Yaskawa INFORM job: R2_O57-69(2)(90,180)OLD.JBI

/JOB
//NAME R2_O57-69(2)(90,180)OLD
//POS
///NPOS 642,642,642,18,0,0
///TOOL 0
///POSTYPE PULSE
///PULSE
C00000=-118942,38116,3308,-51577,58996,23781
C00001=-120746,43281,8706,-50981,57603,23623
C00002=-121445,45407,10966,-50768,57038,23575
C00003=-122175,45836,11424,-50421,56611,23420
C00004=-121445,45407,10966,-50768,57038,23575
C00005=-119713,46835,12049,-51615,58009,23970
C00006=-119593,49070,14464,-51837,57860,24140
C00007=-119713,46835,12049,-51615,58009,23970
C00008=-119003,44749,9818,-51825,58584,24014
C00009=-117170,39689,4492,-52413,60002,24162
C00010=-133704,84336,30677,-4045,90342,4182
C00011=-133972,88781,39264,-3963,87336,4193
C00012=-134077,90756,42954,-3934,86079,4199
C00013=-134077,90297,43636,-3936,85425,4220
C00014=-134077,90756,42954,-3934,86079,4199
C00015=-134064,91533,43556,-3938,86108,4203
C00016=-134173,94225,46985,-3908,85378,4191
C00017=-134064,91533,43556,-3938,86108,4203
C00018=-133960,89550,39850,-3967,87371,4196
C00019=-133691,85093,31233,-4049,90389,4184
C00020=-133097,85072,31507,-9968,91856,10528
C00021=-133756,89066,39535,-9767,88935,10550
C00022=-134013,90847,42981,-9696,87717,10563
C00023=-134013,90387,43661,-9698,87071,10613
C00024=-134013,90847,42981,-9696,87717,10563
C00025=-134077,91446,43535,-9678,87677,10545
C00026=-134345,93924,46689,-9607,86989,10512
C00027=-134077,91446,43535,-9678,87677,10545
C00028=-133821,89654,40071,-9749,88900,10532
C00029=-133165,85640,32010,-9949,91831,10509
C00030=-130607,9372,-15044,-13437,81583,13219
C00031=-132164,5171,-3952,-15307,72023,14325
C00032=-104612,24784,65967,-49840,36559,34272
C00033=-106530,34976,78845,-52404,33899,35280
C00034=-107268,39847,85132,-53931,32696,35940
C00035=-107268,43497,90995,-56192,31674,37136
C00036=-107268,39847,85132,-53931,32696,35940
C00037=-106991,38998,84230,-53831,32905,35947
C00038=-107592,41782,87346,-54342,32315,36087
C00039=-106991,38998,84230,-53831,32905,35947
C00040=-106248,34218,78071,-52358,34091,35316
C00041=-104315,24157,65380,-49864,36729,34346
C00042=-95633,-69755,-51009,-37313,58213,27375
C00043=-82988,-118583,-84497,-42047,60487,32680
C00044=-200995,-130184,-93319,70720,78040,-43840
C00045=-163099,-71600,-71646,60941,59675,-30655
C00046=-151416,29115,15831,69500,88499,-38418
C00047=-148764,29488,16198,69305,86698,-38096
C00048=-147706,29711,16418,69221,85978,-37969
C00049=-147097,31186,17883,69177,85514,-37952
C00050=-147706,29711,16418,69221,85978,-37969
C00051=-147508,26891,13470,69190,85984,-37787
C00052=-146989,25154,11784,69139,85690,-37658
C00053=-147508,26891,13470,69190,85984,-37787
C00054=-148579,26663,13248,69280,86712,-37916
C00055=-151265,26278,12874,69491,88533,-38244
C00056=-151230,28714,15393,69487,88397,-38368
C00057=-148574,29104,15777,69288,86594,-38045
C00058=-147514,29335,16004,69203,85873,-37918
C00059=-146906,30812,17468,69159,85409,-37901
C00060=-147514,29335,16004,69203,85873,-37918
C00061=-147724,26972,13590,69210,86117,-37828
C00062=-147207,25230,11899,69159,85824,-37699
C00063=-147724,26972,13590,69210,86117,-37828
C00064=-148795,26752,13377,69299,86844,-37957
C00065=-151480,26388,13023,69506,88665,-38286
C00066=-150499,113686,46157,71277,96983,-27560
C00067=-148414,114188,46840,70516,95698,-27414
C00068=-147582,114456,47206,70210,95177,-27363
C00069=-147103,116179,49560,69975,94689,-27557
C00070=-147582,114456,47206,70210,95177,-27363
C00071=-147564,110815,41655,70398,95727,-26688
C00072=-147157,108917,39076,70325,95714,-26378
C00073=-147564,110815,41655,70398,95727,-26688
C00074=-148407,110561,41310,70722,96244,-26740
C00075=-150520,110089,40669,71527,97523,-26888
C00076=-135781,-39109,-42450,-5820,71469,-27792
C00077=-134852,-34609,-36187,-6165,70004,-27387
C00078=-134494,-32781,-33633,-6302,69403,-27227
C00079=-134494,-32513,-32201,-6332,68664,-27188
C00080=-134494,-32781,-33633,-6302,69403,-27227
C00081=-134576,-33268,-34172,-6273,69478,-27261
C00082=-134372,-31123,-32745,-6329,69716,-27200
C00083=-134576,-33268,-34172,-6273,69478,-27261
C00084=-133492,-33488,-34057,-6622,69381,-26865
C00085=-132368,-33840,-34288,-6976,69438,-26463
C00086=-133492,-33488,-34057,-6622,69381,-26865
C00087=-133841,-35331,-36614,-6487,69976,-27023
C00088=-134747,-39871,-42887,-6148,71424,-27423
C00089=-122053,-39806,-42652,-15420,62809,-34817
C00090=-121499,-35034,-36226,-15868,61466,-34410
C00091=-121286,-33103,-33607,-16052,60912,-34244
C00092=-121286,-32828,-32171,-16165,60197,-34138
C00093=-121286,-33103,-33607,-16052,60912,-34244
C00094=-121314,-33263,-34344,-15985,61264,-34307
C00095=-121302,-31081,-32892,-15957,61485,-34335
C00096=-121314,-33263,-34344,-15985,61264,-34307
C00097=-119787,-33398,-34061,-16683,61335,-33713
C00098=-118651,-33362,-34037,-17169,61575,-33298
C00099=-119787,-33398,-34061,-16683,61335,-33713
C00100=-119983,-35334,-36680,-16506,61888,-33874
C00101=-120494,-40120,-43107,-16077,63224,-34271
C00102=-114895,-27674,-41035,-24554,79329,-24611
C00103=-103160,-731,-14280,-43401,100853,-1823
C00104=-105135,1502,-9443,-43163,98538,-1741
C00105=-105913,2477,-7430,-43084,97612,-1705
C00106=-105914,2666,-6021,-42996,97041,-1463
C00107=-105913,2477,-7430,-43084,97612,-1705
C00108=-127520,-68112,-41549,-19229,27618,7061
C00109=-127380,-66019,-40542,-19113,28083,7011
C00110=-127520,-68112,-41549,-19229,27618,7061
C00111=-133514,-23938,-39247,-1523,83124,-19162
C00112=-132464,-24298,-39502,-1762,83117,-18812
C00113=-133514,-23938,-39247,-1523,83124,-19162
C00114=-133840,-25466,-41668,-1447,83823,-19278
C00115=-134685,-29188,-47604,-1253,85549,-19576
C00116=-94540,-44906,-54644,-54690,80182,11416
C00117=-2997,-159102,-96620,-35577,110249,43089
C00118=-94928,-31896,-36448,-44981,51726,73410
C00119=-97674,-28950,-32085,-44251,49500,73032
C00120=-98746,-27702,-30280,-43966,48623,72882
C00121=-98747,-27457,-28859,-44425,48077,73195
C00122=-98746,-27702,-30280,-43966,48623,72882
C00123=-99145,-25229,-28534,-43633,48570,72671
C00124=-99641,-23313,-27181,-43273,48438,72445
C00125=-99145,-25229,-28534,-43633,48570,72671
C00126=-99389,-27279,-29944,-43614,48313,72668
C00127=-100362,-28273,-30629,-43136,47769,72383
C00128=-99389,-27279,-29944,-43614,48313,72668
C00129=-98324,-28543,-31764,-43902,49185,72819
C00130=-95596,-31533,-36163,-44641,51397,73201
C00131=-73206,-49255,-47301,-54380,62174,80035
C00132=-83647,-21856,-29546,-43638,51559,72523
C00133=-86196,-18896,-25023,-42989,49379,72216
C00134=-87192,-17643,-23150,-42742,48516,72095
C00135=-87193,-17430,-21742,-43197,47953,72406
C00136=-87192,-17643,-23150,-42742,48516,72095
C00137=-87217,-17769,-23202,-42747,48480,72100
C00138=-88162,-16936,-22585,-42189,48060,71766
C00139=-87217,-17769,-23202,-42747,48480,72100
C00140=-86221,-19023,-25076,-42995,49342,72221
C00141=-83670,-21988,-29600,-43645,51522,72530
C00142=-60313,-109588,-73152,-60260,62863,-74993
C00143=-60313,-109588,-73152,-60260,62863,-74993
C00144=-60313,-109588,-73152,-60260,62863,-74993
C00145=-60313,-109588,-73152,-60260,62863,-74993
C00146=-121468,-98128,-128632,1200,91954,-4785
C00147=-120935,-89040,-122262,1025,92698,-4621
C00148=-120739,-85841,-119804,961,92827,-4562
C00149=-120740,-85741,-118114,960,91838,-4570
C00150=-120739,-85841,-119804,961,92827,-4562
C00151=-120638,-81288,-118578,930,94411,-4521
C00152=-120241,-74983,-116497,803,96366,-4393
C00153=-120638,-81288,-118578,930,94411,-4521
C00154=-120828,-84219,-120984,993,94387,-4576
C00155=-121344,-92430,-127180,1163,93987,-4729
C00156=-126619,-93375,-85777,19436,85602,-57728
C00157=-123229,-93449,-82463,19138,82838,-56953
C00158=-121861,-93330,-81074,19019,81766,-56629
C00159=-121850,-91527,-78779,19037,81304,-56698
C00160=-121861,-93330,-81074,19019,81766,-56629
C00161=-120032,-93477,-81181,18813,81333,-56039
C00162=-117985,-95044,-81508,18598,80291,-55463
C00163=-120032,-93477,-81181,18813,81333,-56039
C00164=-121407,-93650,-82591,18940,82390,-56369
C00165=-124815,-93717,-85961,19254,85118,-57161
C00166=-105133,-95150,-84366,-27685,77771,48864
C00167=-109419,-93151,-80804,-27043,75322,47788
C00168=-111110,-92231,-79325,-26774,74383,47352
C00169=-111209,-90435,-77025,-26813,73909,47425
C00170=-111110,-92231,-79325,-26774,74383,47352
C00171=-111989,-92454,-79471,-26607,74078,47081
C00172=-114284,-92810,-79614,-26159,73263,46376
C00173=-111989,-92454,-79471,-26607,74078,47081
C00174=-110299,-93409,-80962,-26883,75006,47521
C00175=-106012,-95496,-84557,-27540,77427,48607
C00176=-111909,-102425,-108765,-17811,80188,32257
C00177=-116710,-109323,-114600,-10394,73642,20182
C00178=-119128,-100378,-108798,-9411,74366,19294
C00179=-120024,-97049,-106503,-9050,74562,18974
C00180=-120031,-96065,-104948,-9065,74116,19005
C00181=-120024,-97049,-106503,-9050,74562,18974
C00182=-121130,-95394,-105931,-8599,74938,18572
C00183=-122871,-95322,-105904,-7915,74788,17994
C00184=-121130,-95394,-105931,-8599,74938,18572
C00185=-120110,-94835,-105770,-8990,75231,18895
C00186=-120119,-91118,-104720,-8941,76480,18801
C00187=-120110,-94835,-105770,-8990,75231,18895
C00188=-119227,-98081,-108057,-9343,75070,19206
C00189=-116847,-106779,-113833,-10301,74448,20066
C00190=-125162,-107696,-115002,11574,77940,-27023
C00191=-122232,-100471,-109587,10556,77926,-26035
C00192=-121132,-97724,-107430,10172,77873,-25669
C00193=-121129,-96411,-105359,10192,77282,-25717
C00194=-121132,-97724,-107430,10172,77873,-25669
C00195=-120375,-94991,-106195,9888,78418,-25371
C00196=-118057,-94902,-106157,9076,78179,-24616
C00197=-120375,-94991,-106195,9888,78418,-25371
C00198=-121123,-94352,-106931,10125,79277,-25551
C00199=-121107,-89294,-105478,10075,80954,-25409
C00200=-121123,-94352,-106931,10125,79277,-25551
C00201=-122203,-96975,-109071,10499,79378,-25901
C00202=-125076,-103844,-114435,11488,79527,-26845
C00203=-120615,-96693,-99705,24269,61927,-46070
C00204=-120615,-96754,-97435,24583,60621,-46372
C00205=-120615,-96734,-96510,24712,60111,-46493
C00206=-120613,-97925,-98139,24620,60467,-46408
C00207=-122356,-96694,-96496,25580,60643,-47091
C00208=-120617,-95462,-105609,23301,89319,-42487
C00209=-120616,-96376,-102090,23303,86889,-42960
C00210=-120616,-96174,-102896,20314,113785,-36834
C00211=-120616,-95912,-104039,20462,114573,-36686
C00212=-120617,-94981,-106794,20878,116613,-36292
C00213=-120641,-102950,-117078,-2305,90642,6155
C00214=-120615,-96500,-96704,-24731,54164,47412
C00215=-120614,-96434,-94585,-25118,53008,47710
C00216=-120614,-96374,-93724,-25277,52554,47829
C00217=-118876,-96339,-93708,-26332,53098,48481
C00218=-120612,-97606,-95370,-25157,52900,47739
C00219=-120617,-94939,-106140,-23447,89820,42327
C00220=-120616,-95118,-105679,-23443,89475,42395
C00221=-120617,-94553,-107144,-21169,116976,36148
C00222=-120617,-94008,-108179,-21364,117834,35974
C00223=-120617,-92305,-110644,-21913,120064,35505
C00224=-120658,-79064,-115821,-20777,115116,36511
C00225=-120619,-89788,-115023,8813,72744,77332
C00226=-120618,-92923,-112261,8977,69472,77088
C00227=-120618,-93918,-111063,9048,68239,76994
C00228=-120616,-94647,-112535,9016,68763,77035
C00229=-120317,-89862,-109879,8813,69547,77195
C00230=-120618,-93982,-110933,9081,68131,76955
C00231=-120618,-94046,-110802,9114,68024,76915
C00232=-120618,-94709,-109820,9197,65184,76768
C00233=-120617,-95196,-108972,8506,62672,76659
C00234=-120617,-95481,-108396,7103,60843,76635
C00235=-120617,-95545,-108232,5697,60110,76679
C00236=-120618,-93518,-111355,4944,62938,76697
C00237=-120618,-93446,-111427,4025,62977,76727
C00238=-120618,-93195,-111705,2442,63558,76792
C00239=-120618,-92705,-112237,841,64979,76863
C00240=-120618,-92008,-112941,-348,67067,76917
C00241=-120618,-91373,-113529,-886,68931,76945
C00242=-120619,-90404,-114488,-945,70932,76821
C00243=-120619,-89573,-115103,-879,73169,76864
C00244=-120619,-88566,-115779,-154,75847,76963
C00245=-120619,-87861,-116220,1182,77795,77117
C00246=-120619,-87671,-116345,2465,78546,77256
C00247=-120619,-91363,-113807,3286,75243,77100
C00248=-120619,-91437,-113755,4139,75204,77156
C00249=-120618,-91668,-113564,5199,74797,77209
C00250=-120618,-91861,-113400,6010,74299,77242
C00251=-120618,-92325,-112970,7121,73103,77250
C00252=-120618,-92854,-112432,8036,71559,77218
C00253=-120618,-93200,-112056,8504,70412,77180
C00254=-120618,-93741,-111409,8966,68528,77095
C00255=-120618,-93842,-111215,9015,68365,77035
C00256=-120618,-93908,-111085,9047,68257,76996
C00257=-120618,-92911,-112281,8976,69491,77090
C00258=-120619,-89769,-115041,8812,72765,77333
C00259=-120613,-94111,-83344,23310,76872,-48529
C00260=-120612,-93123,-79966,23449,75424,-48818
C00261=-120612,-92685,-78593,23509,74854,-48933
C00262=-120519,-94136,-80334,23460,75127,-48843
C00263=-122104,-91474,-78326,23730,75702,-49326
C00264=-117316,-93808,-82805,15952,85371,-55800
C00265=-120612,-92504,-78008,16222,83828,-57165
C00266=-120612,-92225,-77144,16221,83447,-57214
C00267=-120612,-92754,-78742,16205,84132,-57123
C00268=-120612,-93939,-82668,16176,85870,-56895
C00269=-114287,-94620,-89520,-6331,89004,4508
C00270=-108926,-90943,-77088,-25317,82681,56680
C00271=-112815,-90510,-73836,-25087,79880,55819
C00272=-114383,-90199,-72475,-24991,78788,55461
C00273=-114333,-91608,-74232,-24970,79128,55408
C00274=-112663,-89963,-72378,-25142,79365,55987
C00275=-114583,-88799,-68791,-27921,64605,46597
C00276=-114487,-93503,-82637,-26827,70088,45260
C00277=-115264,-91797,-76742,-30984,57662,33422
C00278=-113792,-91904,-77552,-31424,58590,33801
C00279=-110138,-91921,-79470,-32448,60976,34690
C00280=-60313,-109588,-73152,-60260,62863,-74993
C00281=-60313,-109588,-73152,-60260,62863,-74993
C00282=-60313,-109588,-73152,-60260,62863,-74993
C00283=-60313,-109588,-73152,-60260,62863,-74993
C00284=-93056,-22452,-26427,-62683,51364,-68554
C00285=-94918,-23815,-27400,-62098,50128,-68890
C00286=-95672,-24335,-27768,-61852,49629,-69030
C00287=-95671,-24543,-29165,-61297,50004,-69420
C00288=-95119,-26190,-29068,-62168,49906,-68831
C00289=-113833,-31923,-32981,-19338,22123,-69808
C00290=-113432,-31852,-32933,-20038,22233,-69480
C00291=-111211,-31381,-32618,-29195,23933,-65184
C00292=-107573,-30332,-31913,-37350,26359,-61322
C00293=-106073,-29797,-31550,-41773,28129,-59204
C00294=-102671,-28354,-30566,-47316,31086,-56518
C00295=-101245,-27653,-30084,-50385,33119,-55008
C00296=-96015,-24564,-27929,-57391,39606,-51469
C00297=-95870,-24466,-27860,-57479,39693,-51427
C00298=-98425,-26093,-29002,-49127,35298,-40867
C00299=-98535,-26162,-29051,-49050,35234,-40906
C00300=-98812,-26334,-29170,-48853,35075,-41005
C00301=-94260,-52437,-45641,-55679,35604,-37348
C00302=-53363,-13156,-19582,-69042,101484,-57693
C00303=-70300,5852,-4038,-68507,90193,-60008
C00304=-72032,2742,-6705,-68392,89052,-60255
C00305=-72741,1528,-7732,-68341,88581,-60353
C00306=-72740,1358,-9123,-68348,88884,-60681
C00307=-71868,858,-8294,-68404,89165,-60238
C00308=-77282,-5546,-13564,-65427,71560,-48018
C00309=-76174,-3931,-12256,-66124,74358,-47138
C00310=-77728,-6177,-14071,-64696,69365,-41232
C00311=-76987,-5122,-13221,-65187,71135,-40572
C00312=-78162,-6780,-14553,-64908,67376,-44626
C00313=-76574,-4519,-12734,-65439,69183,-44207
C00314=-75699,-3215,-11672,-66019,71276,-43722
C00315=-73856,-322,-9283,-66697,73982,-43118
C00316=-73074,967,-8204,-67155,75992,-42677
C00317=-72162,2519,-6894,-67667,78480,-42145
C00318=-70374,5730,-4143,-68213,81550,-41494
C00319=-70642,5234,-4572,-68092,80748,-41661
C00320=-70220,6012,-3899,-68142,81024,-41598
C00321=-69181,7983,-2180,-68262,81700,-41439
C00322=-53363,-13156,-19582,-69042,101484,-57693
C00323=-88855,-179547,-122665,-16422,45831,14756
C00324=-103013,-99268,-100595,-7137,71031,6353
C00325=-111832,16928,28851,-4518,50540,4019
C00326=-112106,24952,39258,-4538,48250,4007
C00327=-112211,28376,43752,-4558,47241,4009
C00328=-112092,25909,41315,-4600,47479,4051
C00329=-112213,27385,41422,-4491,48163,3964
C00330=-110994,29129,44722,-10026,47870,8913
C00331=-107882,31558,47633,-16852,48960,15049
C00332=-106420,34221,50265,-20220,50689,15733
C00333=-107556,33681,49588,-20659,51389,16328
C00334=-107303,34756,50847,-23620,53119,19537
C00335=-105809,38630,55063,-26127,54547,25185
C00336=-100600,65185,87794,-37926,61057,39597
C00337=-99799,61843,82703,-37497,62519,39384
C00338=-97770,55081,72181,-36715,65773,39058
C00339=-113055,9147,22486,-11521,49710,9806
C00340=-113748,16710,31984,-11522,47692,9742
C00341=-114014,19893,36035,-11546,46813,9730
C00342=-113504,17960,34216,-11778,47009,9938
C00343=-114013,18924,33775,-11384,47689,9622
C00344=-106504,35034,50196,-27270,57817,24489
C00345=-107808,31596,46678,-26860,57759,23943
C00346=-101619,66436,89448,-39641,65847,43373
C00347=-100773,63725,85128,-39270,67197,43204
C00348=-98646,58275,76145,-38555,70253,42947
C00349=-99884,14179,20835,-32070,74790,34547
C00350=-104259,-119010,-113397,-13066,68419,11198
C00351=-100618,-153040,-123102,-15914,57898,13971
C00352=-171047,-67517,-68920,2824,104590,-81494
C00353=-162612,-44481,-56179,3922,108231,-78415
C00354=-172950,15898,5057,-12161,117913,80240
C00355=-173383,11030,3410,-12137,116393,80239
C00356=-173563,9131,2831,-12130,115759,80238
C00357=-174118,10117,2984,-12376,116079,79984
C00358=-173005,10826,4333,-11924,115790,80453
C00359=-173900,36762,39678,-14923,122347,88654
C00360=-174631,19304,16630,-12631,116903,82099
C00361=-174582,11977,8086,-12295,113872,80049
C00362=-174393,13825,8643,-12294,114494,80054
C00363=-173937,18573,10240,-12297,115988,80066
C00364=-161354,27343,19699,-12039,109597,67520
C00365=-162299,23506,18954,-12170,107974,67338
C00366=-162689,22031,18738,-12226,107304,67264
C00367=-162689,21613,17076,-12289,108094,67181
C00368=-162258,23995,20616,-12099,107225,67431
C00369=-160599,18374,15454,-16346,104951,65883
C00370=-160862,19037,16144,-16128,105227,62268
C00371=-158963,16179,14200,-19810,103313,58208
C00372=-158332,17222,14010,-19745,104082,58313
C00373=-156794,20003,13731,-19594,105963,58572
C00374=-161333,16594,8144,-10689,103467,-23902
C00375=-160995,17911,13523,-10509,100921,-23559
C00376=-160860,18544,15785,-10444,99888,-23423
C00377=-160126,17389,14600,-10331,100117,-23184
C00378=-160925,18232,14234,-10487,100661,-23512
C00379=-160747,19067,16273,-10425,99872,-23382
C00380=-160882,18430,14006,-10490,100906,-23518
C00381=-161218,17106,8616,-10669,103455,-23860
C00382=-159736,50763,37041,-6948,117736,-78214
C00383=-159788,45167,33757,-6909,116883,-78180
C00384=-159810,42990,32553,-6892,116506,-78165
C00385=-160346,43786,32675,-7123,116791,-78393
C00386=-159444,45178,34878,-6729,116233,-78006
C00387=-161348,81543,87740,-6707,117550,-69501
C00388=-161230,54566,49708,-6566,116296,-76295
C00389=-160797,45806,38282,-7135,114356,-78411
C00390=-160766,47971,39500,-7147,114719,-78422
C00391=-160691,53556,42838,-7172,115535,-78445
C00392=-154706,39789,27555,-8539,114606,12724
C00393=-148495,53758,55593,-7913,102792,72747
C00394=-149088,49534,53986,-8041,101563,72620
C00395=-149332,47922,53457,-8093,101041,72570
C00396=-149332,46980,51118,-8127,101987,72507
C00397=-149055,50602,56404,-8000,100635,72693
C00398=-147241,44754,50188,-12563,99747,71321
C00399=-147513,45427,50986,-12280,99912,67703
C00400=-145634,43287,49424,-16194,98869,63733
C00401=-145156,44506,49535,-16105,99500,63818
C00402=-143994,47742,50063,-15894,101016,64033
C00403=-161265,51089,39840,-10591,101724,-23724
C00404=-160975,52973,46100,-10427,98924,-23381
C00405=-160859,53890,48805,-10368,97764,-23243
C00406=-160229,52461,47107,-10276,98151,-23055
C00407=-160915,53398,46988,-10405,98609,-23333
C00408=-160762,54537,49526,-10349,97667,-23200
C00409=-160878,53605,46802,-10407,98831,-23339
C00410=-161167,51693,40503,-10570,101641,-23682
C00411=-148526,37088,19319,-8739,116408,71765
C00412=-149143,32311,17412,-8825,115075,71633
C00413=-149398,30453,16735,-8860,114515,71580
C00414=-149398,30263,15299,-8924,115292,71518
C00415=-149109,32604,18884,-8755,114332,71704
C00416=-147222,27780,14258,-13593,112811,69882
C00417=-147505,28304,14841,-13306,113042,66284
C00418=-145549,26214,13499,-17411,111682,61933
C00419=-145053,27746,13857,-17364,112331,62024
C00420=-143846,31723,14951,-17251,113896,62249
C00421=-164842,-38441,-59879,14258,84390,68161
C00422=-159089,-119441,-87904,20108,53110,65909
C00423=-167794,-136231,-92390,25307,50039,61231
C00424=-105945,-102671,-115440,26558,80933,-73598
C00425=-110364,-40123,-85663,27999,94589,-71935
C00426=-95866,64314,90102,38927,85041,-69053
C00427=-95118,63196,89692,39138,84476,-68962
C00428=-95722,60422,85500,38938,85635,-68779
C00429=-95367,67809,95356,39124,83704,-69344
C00430=-95389,64313,91842,39100,84004,-69244
C00431=-93119,49699,70965,34888,83296,-74684
C00432=-91573,45828,64995,32087,82929,-76236
C00433=-92175,46461,64458,31959,83708,-76245
C00434=-93644,48287,63421,31668,85593,-76279
C00435=-107566,-14252,9731,28298,67477,41115
C00436=-107311,-10314,17293,28810,65069,40577
C00437=-107211,-8617,20467,29042,64083,40348
C00438=-106149,-8342,20561,28950,63805,40701
C00439=-107303,-9723,18207,28865,64837,40517
C00440=-107260,-8071,20895,29042,64114,40337
C00441=-107361,-9770,17714,28809,65103,40566
C00442=-107614,-13711,10138,28297,67517,41106
C00443=-102856,-73680,-76596,22146,63215,42111
C00444=-159709,-90647,-84021,39939,81385,24012
C00445=-89629,-138278,-77876,-2613,32114,-4559
C00446=-116866,-116923,-63332,14121,27231,-27701
C00447=-115505,-113884,-61604,12498,27509,-26695
C00448=-115326,-115959,-62110,12631,26745,-26737
C00449=-117688,-114707,-62647,14613,28063,-28063
C00450=-116558,-113464,-61851,14335,28746,-26693
C00451=-118841,-112467,-62256,17923,31430,-26552
C00452=-113340,-111890,-64159,7172,33609,-21208
C00453=-114395,-115039,-66037,8124,33246,-21857
C00454=-122649,-85452,-63239,9213,34716,17761
C00455=-134041,-32885,-33620,13278,27002,71259
C00456=-134041,-32878,-33615,13278,27003,71259
C00457=-134041,-32875,-33613,13278,27003,71259
C00458=-134243,-35023,-35024,13683,26807,71061
C00459=-134041,-33117,-35025,12952,27729,71423
C00460=-134039,-32852,-33598,169,25633,78300
C00461=-134039,-32854,-33600,1649,26450,70781
C00462=-134033,-32782,-33552,-26231,28846,72528
C00463=-134032,-32780,-33551,-26232,28846,72529
C00464=-134031,-32775,-33547,-26233,28847,72529
C00465=-134045,-33787,-47185,-21244,36087,69888
C00466=-134041,-32886,-33621,13278,27002,71259
C00467=-134041,-32878,-33616,13278,27003,71259
C00468=-134041,-32875,-33614,13278,27003,71259
C00469=-134243,-35024,-35024,13684,26807,71061
C00470=-134041,-33118,-35026,12952,27729,71423
C00471=-134039,-32851,-33598,169,25633,78300
C00472=-134038,-32847,-33595,-898,26468,70800
C00473=-134033,-32781,-33552,-26231,28846,72528
C00474=-134032,-32780,-33550,-26232,28846,72529
C00475=-134031,-32775,-33547,-26233,28847,72529
C00476=-134033,-32807,-33569,-26308,35204,-51674
C00477=-134033,-32800,-33564,-26308,35204,-51674
C00478=-134033,-32797,-33562,-26308,35205,-51674
C00479=-134234,-34945,-34973,-26254,34929,-51698
C00480=-134032,-33039,-34974,-25852,35877,-51926
C00481=-134031,-32780,-33551,-33925,38137,-46837
C00482=-134030,-32755,-33534,-40499,34489,-51688
C00483=-134024,-32674,-33480,-63182,37461,-51745
C00484=-134024,-32672,-33479,-63182,37461,-51745
C00485=-134023,-32667,-33476,-63182,37462,-51745
C00486=-132274,-93805,-93411,-10969,51655,-47542
C00487=-128603,-177588,-92922,79935,27094,-30929
C00488=-220712,-98286,-76285,54391,96146,-31963
C00489=-184952,-63059,-48640,55161,75645,-24408
C00490=-160799,-33037,-33731,39953,86010,-17371
C00491=-160797,-33031,-33727,39953,86010,-17370
C00492=-161372,-34916,-34964,40000,86113,-17582
C00493=-161596,-32269,-33940,40001,86782,-17427
C00494=-160797,-33031,-33727,39954,86007,-17369
C00495=-160797,-33031,-33727,39954,86007,-17369
C00496=-160798,-33031,-33727,39953,86010,-17370
C00497=-160800,-33038,-33732,39953,86010,-17371
C00498=-161845,-54729,-47543,46717,77238,-21379
C00499=-134060,-33141,-33790,36180,74127,-10109
C00500=-134059,-33123,-33778,36179,74128,-10108
C00501=-134058,-33115,-33773,36179,74129,-10108
C00502=-134260,-35264,-35181,36258,74021,-10232
C00503=-134971,-32933,-34372,36300,74891,-10239
C00504=-134058,-33116,-33773,36179,74126,-10108
C00505=-134058,-33116,-33773,36179,74126,-10108
C00506=-134059,-33117,-33774,36179,74129,-10108
C00507=-134059,-33124,-33779,36179,74129,-10109
C00508=-134061,-33143,-33791,36180,74127,-10110
C00509=-154603,-70143,-52801,41434,56822,-11271
C00510=-233697,-158912,-98343,45711,85738,-36562
C00511=-192750,-134368,-116228,45795,59274,-21429
C00512=-146286,5957,-20405,4483,81226,-784
C00513=-143087,77833,55626,3655,71235,-21
C00514=-143077,84404,30410,3488,90094,518
C00515=-142973,88921,39083,3455,87079,467
C00516=-142932,90928,42809,3445,85817,446
C00517=-142932,91423,42172,3444,86463,463
C00518=-142895,88300,39491,3433,86507,476
C00519=-141651,91294,43270,3060,85682,850
C00520=-137685,92968,45398,1861,85119,2101
C00521=-140907,91434,44974,10035,83374,-9634
C00522=-141153,89375,41251,10096,84618,-9613
C00523=-141784,84734,32608,10277,87581,-9573
C00524=-134927,82297,28432,-4231,89843,4215
C00525=-135205,86732,36934,-4146,86884,4227
C00526=-135312,88694,40576,-4116,85649,4233
C00527=-135048,86331,37610,-4195,86271,4296
C00528=-135312,89191,39937,-4114,86296,4212
C00529=-131131,97718,51799,-14741,88225,12517
C00530=-134404,91131,43379,-13932,89423,11301
C00531=-135590,89058,40758,-13635,89764,10876
C00532=-135274,87435,37525,-13726,90938,10849
C00533=-134466,83798,29971,-13984,93767,10791
C00534=-124065,29550,-6223,-11945,87688,10852
C00535=-142798,-17443,-24047,-1901,70629,2085
C00536=-128958,-75577,-89763,-14465,60088,17152
C00537=-136794,-169084,-119686,-16507,29987,18519
C00538=-120728,-100182,-87766,90,59287,81758
C00539=-120667,-32765,-33541,61,60559,81782
C00540=-120668,-32752,-33532,62,60561,81781
C00541=-120669,-32746,-33528,62,60561,81781
C00542=-119537,-32735,-33521,-457,60565,82216
C00543=-120668,-32988,-34940,61,61306,81782
C00544=-120669,-32746,-33528,62,60561,81781
C00545=-120668,-32752,-33532,62,60561,81781
C00546=-120667,-32765,-33541,61,60559,81782
C00547=-129245,32742,-1401,19411,96333,49090
C00548=-120680,47311,12786,22923,98876,42875
C00549=-120681,47325,12802,22923,98874,42874
C00550=-120681,47331,12808,22923,98874,42874
C00551=-119944,47335,12813,22855,98676,43099
C00552=-120681,47590,11836,22981,99550,43006
C00553=-120681,47331,12808,22923,98874,42874
C00554=-120681,47325,12802,22923,98874,42874
C00555=-120680,47311,12786,22923,98876,42875
C00556=-120680,47311,12786,22923,98876,42875
C00557=-120681,47325,12802,22923,98874,42874
C00558=-120681,47331,12808,22923,98874,42874
C00559=-119944,47336,12814,22855,98676,43099
C00560=-120681,47591,11836,22981,99550,43006
C00561=-120681,47331,12808,22923,98874,42874
C00562=-120681,47325,12802,22923,98874,42874
C00563=-120680,47311,12786,22923,98876,42875
C00564=-130279,10433,-22592,19638,98058,49014
C00565=-80524,6289,-12410,27994,97930,43132
C00566=-80528,6302,-12399,27994,97931,43130
C00567=-80529,6307,-12395,27994,97931,43130
C00568=-80528,6342,-13609,28061,98610,43296
C00569=-80526,8467,-10508,27990,97885,43120
C00570=-80531,6315,-12388,27994,97932,43129
C00571=-80530,6310,-12392,27994,97931,43130
C00572=-80526,6297,-12403,27994,97930,43131
C00573=-80535,6328,-12377,43448,96376,44223
C00574=-80540,6344,-12363,43448,96378,44221
C00575=-80541,6350,-12357,43448,96378,44221
C00576=-80540,6385,-13571,43530,96942,44464
C00577=-80538,8511,-10470,43443,96339,44205
C00578=-80543,6359,-12350,43448,96379,44220
C00579=-80542,6352,-12355,43448,96378,44221
C00580=-80537,6336,-12370,43448,96376,44222
C00581=-80544,6364,-12345,43448,96379,44220
C00582=-80548,6380,-12331,43448,96381,44219
C00583=-80550,6387,-12325,43449,96382,44218
C00584=-80549,6422,-13539,43530,96945,44461
C00585=-80546,8548,-10438,43443,96342,44203
C00586=-80552,6395,-12318,43449,96383,44218
C00587=-80550,6388,-12324,43449,96382,44218
C00588=-80545,6372,-12338,43448,96380,44220
C00589=-80549,-32984,-33707,19991,70236,-81341
C00590=-80555,-32968,-33696,19993,70239,-81342
C00591=-80557,-32962,-33692,19994,70240,-81343
C00592=-80555,-33203,-35103,19909,70941,-81221
C00593=-80552,-30784,-32238,19966,70451,-81305
C00594=-80559,-32953,-33686,19994,70241,-81344
C00595=-80557,-32960,-33690,19994,70240,-81343
C00596=-80551,-32976,-33701,19992,70237,-81341
C00597=-125854,-89644,-68041,26288,64871,-64769
C00598=-122217,-87418,-63795,25670,62409,-63867
C00599=-120772,-86435,-62049,25411,61450,-63497
C00600=-122467,-86560,-62389,25830,62102,-64046
C00601=-120772,-87141,-63633,25274,62005,-63363
C00602=-120758,-81751,-60100,25140,62542,-63230
C00603=-120623,13667,2850,23403,71928,-61123
C00604=-120620,18086,6907,23432,71720,-61165
C00605=-121318,17638,5194,23528,72676,-61236
C00606=-123068,16745,1131,23791,75052,-61411
C00607=-120718,-27867,-44657,79,69917,81769
C00608=-120718,-26776,-39817,80,67499,81767
C00609=-120718,-26257,-37822,80,66538,81767
C00610=-119640,-26248,-37815,-390,66541,82155
C00611=-120717,-26264,-39071,80,67303,81767
C00612=-120711,-21841,-34695,77,66883,81769
C00613=-120650,35351,15016,51,65678,81791
C00614=-120646,39983,19783,50,65126,81792
C00615=-120646,39364,17506,49,66209,81792
C00616=-120646,38094,12108,48,68878,81793
C00617=-153612,49047,-26707,64498,91487,-5920
C00618=-150845,73512,-5373,83970,104809,-22981
C00619=-148408,73109,-6304,82893,103555,-22712
C00620=-147428,73003,-6607,82452,103054,-22609
C00621=-148001,71831,-8074,82818,103406,-22490
C00622=-147899,74428,-4816,82578,103245,-22804
C00623=-147427,70753,-6502,82114,102851,-23187
C00624=-147419,52988,54716,74155,91161,-44529
C00625=-147419,54934,59518,74064,90572,-45394
C00626=-148397,55452,60255,73932,91188,-45577
C00627=-150832,56999,62397,73569,92700,-46059
C00628=-140884,-18735,-61179,30897,50366,-12566
C00629=-166969,-145030,-119194,68580,44942,-33891
C00630=-67019,-62651,-90572,-74651,91543,29998
C00631=-83550,-70287,-94354,-69578,80547,28976
C00632=-118113,45135,-5383,-53477,62772,21593
C00633=-119958,50028,-441,-52672,61500,21423
C00634=-120673,52033,1622,-52372,60985,21368
C00635=-119997,52892,2576,-52813,61241,21572
C00636=-120945,50067,-548,-52079,61051,21176
C00637=-120674,50894,2938,-52984,60116,21943
C00638=-120681,45616,24506,-62142,51168,29315
C00639=-120681,45856,27254,-63270,50415,30127
C00640=-119967,43661,25064,-63378,50976,30156
C00641=-118123,38369,19893,-63730,52373,30282
BC00000=96554,835601,336095
BC00001=96554,835601,336095
BC00002=96554,835601,336095
BC00003=96554,835601,336095
BC00004=96554,835601,336095
BC00005=96554,835601,336095
BC00006=96554,835601,336095
BC00007=96554,835601,336095
BC00008=96554,835601,336095
BC00009=96554,835601,336095
BC00010=136857,845097,148119
BC00011=136857,845097,148119
BC00012=136857,845097,148119
BC00013=136857,845097,148119
BC00014=136857,845097,148119
BC00015=136857,845097,148119
BC00016=136857,845097,148119
BC00017=136857,845097,148119
BC00018=136857,845097,148119
BC00019=136857,845097,148119
BC00020=127763,840597,147521
BC00021=127763,840597,147521
BC00022=127763,840597,147521
BC00023=127763,840597,147521
BC00024=127763,840597,147521
BC00025=127763,840597,147521
BC00026=127763,840597,147521
BC00027=127763,840597,147521
BC00028=127763,840597,147521
BC00029=127763,840597,147521
BC00030=128190,841552,377812
BC00031=128540,842336,416238
BC00032=133280,852949,478773
BC00033=133280,852949,478773
BC00034=133280,852949,478773
BC00035=133280,852949,478773
BC00036=133280,852949,478773
BC00037=133280,852949,478773
BC00038=133280,852949,478773
BC00039=133280,852949,478773
BC00040=133280,852949,478773
BC00041=133280,852949,478773
BC00042=133280,852949,478773
BC00043=133280,740797,478773
BC00044=339531,724265,78042
BC00045=339531,836404,78042
BC00046=339531,836404,78042
BC00047=339531,836404,78042
BC00048=339531,836404,78042
BC00049=339531,836404,78042
BC00050=339531,836404,78042
BC00051=339531,836404,78042
BC00052=339531,836404,78042
BC00053=339531,836404,78042
BC00054=339531,836404,78042
BC00055=339531,836404,78042
BC00056=339904,835618,355430
BC00057=339904,835618,355430
BC00058=339904,835618,355430
BC00059=339904,835618,355430
BC00060=339904,835618,355430
BC00061=339904,835618,355430
BC00062=339904,835618,355430
BC00063=339904,835618,355430
BC00064=339904,835618,355430
BC00065=339904,835618,355430
BC00066=360438,779454,158640
BC00067=360438,779454,158640
BC00068=360438,779454,158640
BC00069=360438,779454,158640
BC00070=360438,779454,158640
BC00071=360438,779454,158640
BC00072=360438,779454,158640
BC00073=360438,779454,158640
BC00074=360438,779454,158640
BC00075=360438,779454,158640
BC00076=287078,719990,246987
BC00077=287078,719990,246987
BC00078=287078,719990,246987
BC00079=287078,719990,246987
BC00080=287078,719990,246987
BC00081=287078,719990,246987
BC00082=287078,719990,246987
BC00083=287078,719990,246987
BC00084=287078,719990,246987
BC00085=287078,719990,246987
BC00086=287078,719990,246987
BC00087=287078,719990,246987
BC00088=287078,719990,246987
BC00089=265919,739566,219094
BC00090=265919,739566,219094
BC00091=265919,739566,219094
BC00092=265919,739566,219094
BC00093=265919,739566,219094
BC00094=265919,739566,219094
BC00095=265919,739566,219094
BC00096=265919,739566,219094
BC00097=265919,739566,219094
BC00098=265919,739566,219094
BC00099=265919,739566,219094
BC00100=265919,739566,219094
BC00101=265919,739566,219094
BC00102=270629,754825,208138
BC00103=280478,786731,185230
BC00104=280478,786731,185230
BC00105=280478,786731,185230
BC00106=280478,786731,185230
BC00107=280478,786731,185230
BC00108=280478,786731,185230
BC00109=280478,786731,185230
BC00110=280478,786731,185230
BC00111=280478,786731,185230
BC00112=280478,786731,185230
BC00113=280478,786731,185230
BC00114=280478,786731,185230
BC00115=280478,786731,185230
BC00116=280478,786731,185230
BC00117=280478,786731,185230
BC00118=398174,660028,119143
BC00119=398174,660028,119143
BC00120=398174,660028,119143
BC00121=398174,660028,119143
BC00122=398174,660028,119143
BC00123=398174,660028,119143
BC00124=398174,660028,119143
BC00125=398174,660028,119143
BC00126=398174,660028,119143
BC00127=398174,660028,119143
BC00128=398174,660028,119143
BC00129=398174,660028,119143
BC00130=398174,660028,119143
BC00131=398174,660028,119143
BC00132=398174,676680,118838
BC00133=398174,676680,118838
BC00134=398174,676680,118838
BC00135=398174,676680,118838
BC00136=398174,676680,118838
BC00137=398174,676680,118838
BC00138=398174,676680,118838
BC00139=398174,676680,118838
BC00140=398174,676680,118838
BC00141=398174,676680,118838
BC00142=398174,709471,119143
BC00143=398174,709471,1074810
BC00144=398174,709471,1074810
BC00145=398174,709471,1074810
BC00146=57444,909387,1075175
BC00147=57444,909387,1075175
BC00148=57444,909387,1075175
BC00149=57444,909387,1075175
BC00150=57444,909387,1075175
BC00151=57444,909387,1075175
BC00152=57444,909387,1075175
BC00153=57444,909387,1075175
BC00154=57444,909387,1075175
BC00155=57444,909387,1075175
BC00156=387812,761116,1075175
BC00157=387812,761116,1075175
BC00158=387812,761116,1075175
BC00159=387812,761116,1075175
BC00160=387812,761116,1075175
BC00161=387812,761116,1075175
BC00162=387812,761116,1075175
BC00163=387812,761116,1075175
BC00164=387812,761116,1075175
BC00165=387812,761116,1075175
BC00166=398174,759145,1075175
BC00167=398174,759145,1075175
BC00168=398174,759145,1075175
BC00169=398174,759145,1075175
BC00170=398174,759145,1075175
BC00171=398174,759145,1075175
BC00172=398174,759145,1075175
BC00173=398174,759145,1075175
BC00174=398174,759145,1075175
BC00175=398174,759145,1075175
BC00176=333134,819567,1075175
BC00177=279823,869094,1075175
BC00178=279823,869094,1075175
BC00179=279823,869094,1075175
BC00180=279823,869094,1075175
BC00181=279823,869094,1075175
BC00182=279823,869094,1075175
BC00183=279823,869094,1075175
BC00184=279823,869094,1075175
BC00185=279823,869094,1075175
BC00186=279823,869094,1075175
BC00187=279823,869094,1075175
BC00188=279823,869094,1075175
BC00189=279823,869094,1075175
BC00190=275316,868895,1075175
BC00191=275316,868895,1075175
BC00192=275316,868895,1075175
BC00193=275316,868895,1075175
BC00194=275316,868895,1075175
BC00195=275316,868895,1075175
BC00196=275316,868895,1075175
BC00197=275316,868895,1075175
BC00198=275316,868895,1075175
BC00199=275316,868895,1075175
BC00200=275316,868895,1075175
BC00201=275316,868895,1075175
BC00202=275316,868895,1075175
BC00203=248617,854140,1075175
BC00204=254056,857807,1075175
BC00205=256232,859273,1075175
BC00206=256232,859273,1075175
BC00207=256232,859273,1075175
BC00208=253226,894872,1075175
BC00209=253181,875400,1075175
BC00210=262196,916333,1075175
BC00211=260159,916876,1075175
BC00212=255067,918234,1075175
BC00213=282270,884174,1075175
BC00214=308566,851249,1075175
BC00215=303275,855484,1075175
BC00216=301159,857178,1075175
BC00217=301159,857178,1075175
BC00218=301159,857178,1075175
BC00219=307004,898560,1075175
BC00220=306997,895900,1075175
BC00221=298092,939734,1075175
BC00222=300138,940270,1075175
BC00223=305253,941611,1075175
BC00224=305253,905163,1075175
BC00225=39900,867009,1075175
BC00226=40577,869537,1075175
BC00227=40847,870549,1075175
BC00228=40847,870549,1075175
BC00229=40847,870549,1075175
BC00230=45513,869797,1075175
BC00231=50182,869045,1075175
BC00232=51093,866125,1075175
BC00233=53315,863718,1075175
BC00234=56508,862165,1075175
BC00235=59299,861864,1075175
BC00236=64319,881411,1075175
BC00237=66008,881734,1075175
BC00238=68698,882694,1075175
BC00239=71220,884421,1075175
BC00240=72871,886722,1075175
BC00241=73248,888700,1075175
BC00242=51462,893621,1075175
BC00243=50596,895819,1075175
BC00244=48515,898291,1075175
BC00245=45388,899920,1075175
BC00246=42604,900254,1075175
BC00247=37204,880652,1075175
BC00248=35531,880431,1075175
BC00249=33623,879614,1075175
BC00250=32102,879156,1075175
BC00251=30367,877607,1075175
BC00252=29250,875773,1075175
BC00253=28488,874624,1075175
BC00254=28403,872555,1075175
BC00255=35406,871426,1075175
BC00256=40072,870674,1075175
BC00257=39801,869663,1075175
BC00258=39125,867134,1075175
BC00259=384225,761552,1075175
BC00260=389728,762459,1075175
BC00261=391929,762822,1075175
BC00262=391929,762822,1075175
BC00263=391929,762822,1075175
BC00264=398174,778803,1075175
BC00265=389293,757453,1075175
BC00266=386948,753680,1075175
BC00267=385197,754103,1075175
BC00268=380821,755163,1075175
BC00269=390241,748582,1075175
BC00270=398174,743040,1075175
BC00271=398174,742992,1075175
BC00272=398174,742973,1075175
BC00273=398174,742973,1075175
BC00274=398174,742973,1075175
BC00275=398174,723539,1075175
BC00276=398174,782754,1075175
BC00277=398174,769979,1075175
BC00278=398174,768078,1075175
BC00279=398174,763325,1075175
BC00280=398174,709471,1074810
BC00281=398174,709471,1074810
BC00282=398174,709471,1074810
BC00283=398174,709471,119143
BC00284=398174,653220,79650
BC00285=398174,657768,64044
BC00286=398174,659587,57801
BC00287=398174,659587,57801
BC00288=398174,659587,57801
BC00289=398174,647459,52964
BC00290=398174,647641,53011
BC00291=398174,647926,52959
BC00292=398174,649471,52960
BC00293=398174,649897,52959
BC00294=398174,651823,52965
BC00295=398174,652427,52966
BC00296=398174,655956,53049
BC00297=398174,656105,52982
BC00298=398174,657480,59322
BC00299=398174,654990,65562
BC00300=398174,648765,81161
BC00301=398174,648765,81161
BC00302=398174,698385,106592
BC00303=398174,698385,106592
BC00304=398174,700489,89398
BC00305=398174,701330,82521
BC00306=398174,701330,82521
BC00307=398174,701330,82521
BC00308=398174,685598,86909
BC00309=398174,688108,86960
BC00310=398174,685139,87079
BC00311=398174,686595,87081
BC00312=398174,683738,83198
BC00313=398174,687564,83231
BC00314=398174,689314,83245
BC00315=398174,694269,83287
BC00316=398174,696128,83303
BC00317=398174,698444,83322
BC00318=398174,704331,83441
BC00319=398174,703537,83349
BC00320=398174,701795,90815
BC00321=398174,697441,109481
BC00322=398174,698385,106592
BC00323=110889,752860,366045
BC00324=110889,839896,366045
BC00325=110889,839896,366045
BC00326=110889,839896,366045
BC00327=110889,839896,366045
BC00328=110889,839896,366045
BC00329=110889,839896,366045
BC00330=110889,839896,366045
BC00331=110889,839896,366045
BC00332=110889,839896,366045
BC00333=110889,839896,366045
BC00334=110889,839896,366045
BC00335=110889,839896,366045
BC00336=110889,839896,366045
BC00337=110889,839896,366045
BC00338=110889,839896,366045
BC00339=123028,849105,365775
BC00340=123028,849105,365775
BC00341=123028,849105,365775
BC00342=123028,849105,365775
BC00343=123028,849105,365775
BC00344=123028,849105,365775
BC00345=123028,849105,365775
BC00346=123028,849105,365775
BC00347=123028,849105,365775
BC00348=123028,849105,365775
BC00349=123028,849105,478951
BC00350=123028,849105,365775
BC00351=123028,739623,365775
BC00352=364766,734562,263233
BC00353=364766,820256,263233
BC00354=364766,820256,263233
BC00355=364766,820256,263233
BC00356=364766,820256,263233
BC00357=364766,820256,263233
BC00358=364766,820256,263233
BC00359=364766,820256,263233
BC00360=364766,820256,263233
BC00361=364766,820256,263233
BC00362=364766,820256,263233
BC00363=364766,820256,263233
BC00364=361551,789276,285866
BC00365=361551,789276,285866
BC00366=361551,789276,285866
BC00367=361551,789276,285866
BC00368=361551,789276,285866
BC00369=361551,789276,285866
BC00370=361551,789276,285866
BC00371=361551,789276,285866
BC00372=361551,789276,285866
BC00373=361551,789276,285866
BC00374=348559,761935,339517
BC00375=348559,761935,339517
BC00376=348559,761935,339517
BC00377=348559,761935,339517
BC00378=348559,761935,339517
BC00379=348559,761935,339517
BC00380=348559,761935,339517
BC00381=348559,761935,339517
BC00382=351688,805610,242925
BC00383=351688,805610,242925
BC00384=351688,805610,242925
BC00385=351688,805610,242925
BC00386=351688,805610,242925
BC00387=351688,805610,242925
BC00388=351688,805610,242925
BC00389=351688,805610,242925
BC00390=351688,805610,242925
BC00391=351688,805610,242925
BC00392=341470,796062,300748
BC00393=334931,789951,337755
BC00394=334931,789951,337755
BC00395=334931,789951,337755
BC00396=334931,789951,337755
BC00397=334931,789951,337755
BC00398=334931,789951,337755
BC00399=334931,789951,337755
BC00400=334931,789951,337755
BC00401=334931,789951,337755
BC00402=334931,789951,337755
BC00403=366370,768147,319209
BC00404=366370,768147,319209
BC00405=366370,768147,319209
BC00406=366370,768147,319209
BC00407=366370,768147,319209
BC00408=366370,768147,319209
BC00409=366370,768147,319209
BC00410=366370,768147,319209
BC00411=331816,834270,221049
BC00412=331816,834270,221049
BC00413=331816,834270,221049
BC00414=331816,834270,221049
BC00415=331816,834270,221049
BC00416=331816,834270,221049
BC00417=331816,834270,221049
BC00418=331816,834270,221049
BC00419=331816,834270,221049
BC00420=331816,834270,221049
BC00421=331816,834270,221049
BC00422=331816,834270,221049
BC00423=331816,756487,221049
BC00424=117407,735681,392880
BC00425=117407,830751,392880
BC00426=117407,830751,392880
BC00427=117407,830751,392880
BC00428=117407,830751,392880
BC00429=117407,830751,392880
BC00430=117407,830751,392880
BC00431=117407,830751,392880
BC00432=117407,830751,392880
BC00433=117407,830751,392880
BC00434=117407,830751,392880
BC00435=165039,821153,488226
BC00436=165039,821153,488226
BC00437=165039,821153,488226
BC00438=165039,821153,488226
BC00439=165039,821153,488226
BC00440=165039,821153,488226
BC00441=165039,821153,488226
BC00442=165039,821153,488226
BC00443=165039,821153,488226
BC00444=165039,716440,488226
BC00445=215467,770281,277938
BC00446=224741,780183,239264
BC00447=224741,780183,239264
BC00448=224741,780183,239264
BC00449=224741,780183,239264
BC00450=223863,780189,235036
BC00451=221998,780202,226059
BC00452=221120,780208,221831
BC00453=221120,780208,221831
BC00454=247700,730574,167564
BC00455=284504,661851,92426
BC00456=283683,667271,73580
BC00457=283355,669439,66042
BC00458=283355,669439,66042
BC00459=283355,669439,66042
BC00460=290618,670312,62214
BC00461=290286,670856,65123
BC00462=313229,678202,54724
BC00463=315006,676391,61005
BC00464=319449,671863,76707
BC00465=319449,671863,76707
BC00466=284327,697642,92813
BC00467=283507,703062,73968
BC00468=283179,705230,66430
BC00469=283179,705230,66430
BC00470=283179,705230,66430
BC00471=290806,706102,62601
BC00472=292572,707091,65141
BC00473=313417,713993,55110
BC00474=315194,712182,61391
BC00475=319637,707653,77094
BC00476=316114,745194,120079
BC00477=315294,750614,101234
BC00478=314966,752782,93695
BC00479=314966,752782,93695
BC00480=314966,752782,93695
BC00481=320510,757143,93053
BC00482=324314,754896,65097
BC00483=342454,763314,11126
BC00484=344231,761502,17407
BC00485=348674,756974,33109
BC00486=323892,760985,88013
BC00487=274329,769006,197820
BC00488=274329,769006,197820
BC00489=274329,769006,197820
BC00490=274329,769006,197820
BC00491=275833,771147,192013
BC00492=275833,771147,192013
BC00493=275833,771147,192013
BC00494=274957,771147,187778
BC00495=273093,771160,178799
BC00496=272212,771172,174576
BC00497=270708,769032,180383
BC00498=260156,771352,186850
BC00499=217949,780633,212721
BC00500=221710,785984,198203
BC00501=223214,788124,192396
BC00502=223214,788124,192396
BC00503=223214,788124,192396
BC00504=222366,788125,188295
BC00505=220474,788138,179183
BC00506=219621,788149,175093
BC00507=218116,786009,180900
BC00508=214355,780658,195417
BC00509=248187,774085,196773
BC00510=248187,774085,196773
BC00511=147181,722952,398153
BC00512=147181,822999,398153
BC00513=147181,848170,350595
BC00514=147181,848170,136674
BC00515=147181,848170,136674
BC00516=147181,848170,136674
BC00517=147181,848170,136674
BC00518=147181,848170,136674
BC00519=147181,848170,136674
BC00520=147181,848170,136674
BC00521=147181,848170,136674
BC00522=147181,848170,136674
BC00523=147181,848170,136674
BC00524=129425,844943,138841
BC00525=129425,844943,138841
BC00526=129425,844943,138841
BC00527=129425,844943,138841
BC00528=129425,844943,138841
BC00529=129425,844943,138841
BC00530=129425,844943,138841
BC00531=129425,844943,138841
BC00532=129425,844943,138841
BC00533=129425,844943,138841
BC00534=129425,844943,363048
BC00535=129425,844943,442423
BC00536=129425,844943,365714
BC00537=129425,734036,365714
BC00538=354451,699777,288314
BC00539=354451,699777,288314
BC00540=354450,701134,261853
BC00541=354450,701677,251269
BC00542=354450,701677,251269
BC00543=354450,701677,251269
BC00544=354460,705283,251308
BC00545=354460,704741,261892
BC00546=354461,703383,288353
BC00547=325656,760789,189206
BC00548=317844,776356,162319
BC00549=317841,777049,135545
BC00550=317840,777326,124835
BC00551=317840,777326,124835
BC00552=317840,777326,124835
BC00553=317851,780938,124874
BC00554=317852,780661,135584
BC00555=317854,779968,162358
BC00556=317959,815888,162746
BC00557=317957,816581,135972
BC00558=317956,816858,125263
BC00559=317956,816858,125263
BC00560=317956,816858,125263
BC00561=317966,820442,125301
BC00562=317967,820165,136011
BC00563=317970,819472,162785
BC00564=325656,760789,189206
BC00565=271909,801758,247550
BC00566=272504,801445,220763
BC00567=272743,801320,210049
BC00568=272743,801320,210049
BC00569=272743,801320,210049
BC00570=275997,799496,210023
BC00571=275759,799621,220738
BC00572=275163,799934,247524
BC00573=278580,798061,194815
BC00574=280931,796764,169534
BC00575=281871,796245,159422
BC00576=281871,796245,159422
BC00577=281871,796245,159422
BC00578=285149,794408,159396
BC00579=284209,794927,169508
BC00580=281858,796225,194789
BC00581=293014,822129,195048
BC00582=295365,820832,169767
BC00583=296305,820313,159654
BC00584=296305,820313,159654
BC00585=296305,820313,159654
BC00586=299523,818510,159629
BC00587=298582,819029,169741
BC00588=296232,820326,195022
BC00589=295296,831576,292226
BC00590=297647,830278,266945
BC00591=298588,829759,256833
BC00592=298588,829759,256833
BC00593=298588,829759,256833
BC00594=301865,827922,256807
BC00595=300925,828441,266919
BC00596=298574,829739,292200
BC00597=257702,768621,237124
BC00598=257702,768621,237124
BC00599=257702,768621,237124
BC00600=257702,768621,237124
BC00601=257702,768621,237124
BC00602=257702,768621,237124
BC00603=257702,768621,237124
BC00604=257702,768621,237124
BC00605=257702,768621,237124
BC00606=257702,768621,237124
BC00607=325913,816678,196275
BC00608=325913,816678,196275
BC00609=325913,816678,196275
BC00610=325913,816678,196275
BC00611=325913,816678,196275
BC00612=325913,816678,196275
BC00613=325913,816678,196275
BC00614=325913,816678,196275
BC00615=325913,816678,196275
BC00616=325913,816678,196275
BC00617=339279,834200,140350
BC00618=341210,836731,132272
BC00619=341210,836731,132272
BC00620=341210,836731,132272
BC00621=341210,836731,132272
BC00622=341210,836731,132272
BC00623=341210,836731,132272
BC00624=341210,836731,132272
BC00625=341210,836731,132272
BC00626=341210,836731,132272
BC00627=341210,836731,132272
BC00628=341210,750693,132272
BC00629=341210,703211,132272
BC00630=96167,714371,303257
BC00631=96167,839119,303257
BC00632=96167,839119,303257
BC00633=96167,839119,303257
BC00634=96167,839119,303257
BC00635=96167,839119,303257
BC00636=96167,839119,303257
BC00637=96167,839119,303257
BC00638=96167,839119,303257
BC00639=96167,839119,303257
BC00640=96167,839119,303257
BC00641=96167,839119,303257
EC00000=798156,1112951
EC00001=798156,1112951
EC00002=798156,1112951
EC00003=798156,1112951
EC00004=798156,1112951
EC00005=798156,1112951
EC00006=798156,1112951
EC00007=798156,1112951
EC00008=798156,1112951
EC00009=798156,1112951
EC00010=798156,1112951
EC00011=798156,1112951
EC00012=798156,1112951
EC00013=798156,1112951
EC00014=798156,1112951
EC00015=798156,1112951
EC00016=798156,1112951
EC00017=798156,1112951
EC00018=798156,1112951
EC00019=798156,1112951
EC00020=798156,1112951
EC00021=798156,1112951
EC00022=798156,1112951
EC00023=798156,1112951
EC00024=798156,1112951
EC00025=798156,1112951
EC00026=798156,1112951
EC00027=798156,1112951
EC00028=798156,1112951
EC00029=798156,1112951
EC00030=798156,1112951
EC00031=798156,1112951
EC00032=798156,1112951
EC00033=798156,1112951
EC00034=798156,1112951
EC00035=798156,1112951
EC00036=798156,1112951
EC00037=798156,1112951
EC00038=798156,1112951
EC00039=798156,1112951
EC00040=798156,1112951
EC00041=798156,1112951
EC00042=798156,1112951
EC00043=798156,1112951
EC00044=798156,1112951
EC00045=798156,1112951
EC00046=798156,1112951
EC00047=798156,1112951
EC00048=798156,1112951
EC00049=798156,1112951
EC00050=798156,1112951
EC00051=798156,1112951
EC00052=798156,1112951
EC00053=798156,1112951
EC00054=798156,1112951
EC00055=798156,1112951
EC00056=798156,1112951
EC00057=798156,1112951
EC00058=798156,1112951
EC00059=798156,1112951
EC00060=798156,1112951
EC00061=798156,1112951
EC00062=798156,1112951
EC00063=798156,1112951
EC00064=798156,1112951
EC00065=798156,1112951
EC00066=798156,1112951
EC00067=798156,1112951
EC00068=798156,1112951
EC00069=798156,1112951
EC00070=798156,1112951
EC00071=798156,1112951
EC00072=798156,1112951
EC00073=798156,1112951
EC00074=798156,1112951
EC00075=798156,1112951
EC00076=798156,1112951
EC00077=798156,1112951
EC00078=798156,1112951
EC00079=798156,1112951
EC00080=798156,1112951
EC00081=798156,1112951
EC00082=798156,1112951
EC00083=798156,1112951
EC00084=798156,1112951
EC00085=798156,1112951
EC00086=798156,1112951
EC00087=798156,1112951
EC00088=798156,1112951
EC00089=798156,1112951
EC00090=798156,1112951
EC00091=798156,1112951
EC00092=798156,1112951
EC00093=798156,1112951
EC00094=798156,1112951
EC00095=798156,1112951
EC00096=798156,1112951
EC00097=798156,1112951
EC00098=798156,1112951
EC00099=798156,1112951
EC00100=798156,1112951
EC00101=798156,1112951
EC00102=798156,1112951
EC00103=798156,1112951
EC00104=798156,1112951
EC00105=798156,1112951
EC00106=798156,1112951
EC00107=798156,1112951
EC00108=798156,1112951
EC00109=798156,1112951
EC00110=798156,1112951
EC00111=798156,1112951
EC00112=798156,1112951
EC00113=798156,1112951
EC00114=798156,1112951
EC00115=798156,1112951
EC00116=798156,1112951
EC00117=798156,1112951
EC00118=798156,1112951
EC00119=798156,1112951
EC00120=798156,1112951
EC00121=798156,1112951
EC00122=798156,1112951
EC00123=798156,1112951
EC00124=798156,1112951
EC00125=798156,1112951
EC00126=798156,1112951
EC00127=798156,1112951
EC00128=798156,1112951
EC00129=798156,1112951
EC00130=798156,1112951
EC00131=798156,1112951
EC00132=798156,1112951
EC00133=798156,1112951
EC00134=798156,1112951
EC00135=798156,1112951
EC00136=798156,1112951
EC00137=798156,1112951
EC00138=798156,1112951
EC00139=798156,1112951
EC00140=798156,1112951
EC00141=798156,1112951
EC00142=798156,1112951
EC00143=798156,1112951
EC00144=975524,1112951
EC00145=975524,1112951
EC00146=975524,1112951
EC00147=975524,1112951
EC00148=975524,1112951
EC00149=975524,1112951
EC00150=975524,1112951
EC00151=975524,1112951
EC00152=975524,1112951
EC00153=975524,1112951
EC00154=975524,1112951
EC00155=975524,1112951
EC00156=975524,1112951
EC00157=975524,1112951
EC00158=975524,1112951
EC00159=975524,1112951
EC00160=975524,1112951
EC00161=975524,1112951
EC00162=975524,1112951
EC00163=975524,1112951
EC00164=975524,1112951
EC00165=975524,1112951
EC00166=975524,1112951
EC00167=975524,1112951
EC00168=975524,1112951
EC00169=975524,1112951
EC00170=975524,1112951
EC00171=975524,1112951
EC00172=975524,1112951
EC00173=975524,1112951
EC00174=975524,1112951
EC00175=975524,1112951
EC00176=975524,1112951
EC00177=975524,1112951
EC00178=975524,1112951
EC00179=975524,1112951
EC00180=975524,1112951
EC00181=975524,1112951
EC00182=975524,1112951
EC00183=975524,1112951
EC00184=975524,1112951
EC00185=975524,1112951
EC00186=975524,1112951
EC00187=975524,1112951
EC00188=975524,1112951
EC00189=975524,1112951
EC00190=975524,1112951
EC00191=975524,1112951
EC00192=975524,1112951
EC00193=975524,1112951
EC00194=975524,1112951
EC00195=975524,1112951
EC00196=975524,1112951
EC00197=975524,1112951
EC00198=975524,1112951
EC00199=975524,1112951
EC00200=975524,1112951
EC00201=975524,1112951
EC00202=975524,1112951
EC00203=975524,1112951
EC00204=975524,1112951
EC00205=975524,1112951
EC00206=975524,1112951
EC00207=975524,1112951
EC00208=975524,1112951
EC00209=975524,1112951
EC00210=975524,1112951
EC00211=975524,1112951
EC00212=975524,1112951
EC00213=975524,1112951
EC00214=975524,1112951
EC00215=975524,1112951
EC00216=975524,1112951
EC00217=975524,1112951
EC00218=975524,1112951
EC00219=975524,1112951
EC00220=975524,1112951
EC00221=975524,1112951
EC00222=975524,1112951
EC00223=975524,1112951
EC00224=975524,1112951
EC00225=975524,1112951
EC00226=975524,1112951
EC00227=975524,1112951
EC00228=975524,1112951
EC00229=975524,1112951
EC00230=975524,1112951
EC00231=975524,1112951
EC00232=975524,1112951
EC00233=975524,1112951
EC00234=975524,1112951
EC00235=975524,1112951
EC00236=975524,1112951
EC00237=975524,1112951
EC00238=975524,1112951
EC00239=975524,1112951
EC00240=975524,1112951
EC00241=975524,1112951
EC00242=975524,1112951
EC00243=975524,1112951
EC00244=975524,1112951
EC00245=975524,1112951
EC00246=975524,1112951
EC00247=975524,1112951
EC00248=975524,1112951
EC00249=975524,1112951
EC00250=975524,1112951
EC00251=975524,1112951
EC00252=975524,1112951
EC00253=975524,1112951
EC00254=975524,1112951
EC00255=975524,1112951
EC00256=975524,1112951
EC00257=975524,1112951
EC00258=975524,1112951
EC00259=975524,1112951
EC00260=975524,1112951
EC00261=975524,1112951
EC00262=975524,1112951
EC00263=975524,1112951
EC00264=975524,1112951
EC00265=975524,1112951
EC00266=975524,1112951
EC00267=975524,1112951
EC00268=975524,1112951
EC00269=975524,1112951
EC00270=975524,1112951
EC00271=975524,1112951
EC00272=975524,1112951
EC00273=975524,1112951
EC00274=975524,1112951
EC00275=975524,1112951
EC00276=975524,1112951
EC00277=975524,1112951
EC00278=975524,1112951
EC00279=975524,1112951
EC00280=975524,1112951
EC00281=975524,1112951
EC00282=798156,1112951
EC00283=798156,1112951
EC00284=798156,1112951
EC00285=798156,1112951
EC00286=798156,1112951
EC00287=798156,1112951
EC00288=798156,1112951
EC00289=798156,1112951
EC00290=798156,1112951
EC00291=798156,1112951
EC00292=798156,1112951
EC00293=798156,1112951
EC00294=798156,1112951
EC00295=798156,1112951
EC00296=798156,1112951
EC00297=798156,1112951
EC00298=798156,1112951
EC00299=798156,1112951
EC00300=798156,1112951
EC00301=798156,1112951
EC00302=798156,1112951
EC00303=798156,1112951
EC00304=798156,1112951
EC00305=798156,1112951
EC00306=798156,1112951
EC00307=798156,1112951
EC00308=798156,1112951
EC00309=798156,1112951
EC00310=798156,1112951
EC00311=798156,1112951
EC00312=798156,1112951
EC00313=798156,1112951
EC00314=798156,1112951
EC00315=798156,1112951
EC00316=798156,1112951
EC00317=798156,1112951
EC00318=798156,1112951
EC00319=798156,1112951
EC00320=798156,1112951
EC00321=798156,1112951
EC00322=798156,1112951
EC00323=798156,1112951
EC00324=798156,1112951
EC00325=798156,1112951
EC00326=798156,1112951
EC00327=798156,1112951
EC00328=798156,1112951
EC00329=798156,1112951
EC00330=798156,1112951
EC00331=798156,1112951
EC00332=798156,1112951
EC00333=798156,1112951
EC00334=798156,1112951
EC00335=798156,1112951
EC00336=798156,1112951
EC00337=798156,1112951
EC00338=798156,1112951
EC00339=798156,1112951
EC00340=798156,1112951
EC00341=798156,1112951
EC00342=798156,1112951
EC00343=798156,1112951
EC00344=798156,1112951
EC00345=798156,1112951
EC00346=798156,1112951
EC00347=798156,1112951
EC00348=798156,1112951
EC00349=798156,1112951
EC00350=798156,1112951
EC00351=798156,1112951
EC00352=798156,1112951
EC00353=798156,1112951
EC00354=798156,1112951
EC00355=798156,1112951
EC00356=798156,1112951
EC00357=798156,1112951
EC00358=798156,1112951
EC00359=798156,1112951
EC00360=798156,1112951
EC00361=798156,1112951
EC00362=798156,1112951
EC00363=798156,1112951
EC00364=798156,1112951
EC00365=798156,1112951
EC00366=798156,1112951
EC00367=798156,1112951
EC00368=798156,1112951
EC00369=798156,1112951
EC00370=798156,1112951
EC00371=798156,1112951
EC00372=798156,1112951
EC00373=798156,1112951
EC00374=798156,1112951
EC00375=798156,1112951
EC00376=798156,1112951
EC00377=798156,1112951
EC00378=798156,1112951
EC00379=798156,1112951
EC00380=798156,1112951
EC00381=798156,1112951
EC00382=798156,1112951
EC00383=798156,1112951
EC00384=798156,1112951
EC00385=798156,1112951
EC00386=798156,1112951
EC00387=798156,1112951
EC00388=798156,1112951
EC00389=798156,1112951
EC00390=798156,1112951
EC00391=798156,1112951
EC00392=798156,1112951
EC00393=798156,1112951
EC00394=798156,1112951
EC00395=798156,1112951
EC00396=798156,1112951
EC00397=798156,1112951
EC00398=798156,1112951
EC00399=798156,1112951
EC00400=798156,1112951
EC00401=798156,1112951
EC00402=798156,1112951
EC00403=798156,1112951
EC00404=798156,1112951
EC00405=798156,1112951
EC00406=798156,1112951
EC00407=798156,1112951
EC00408=798156,1112951
EC00409=798156,1112951
EC00410=798156,1112951
EC00411=798156,1112951
EC00412=798156,1112951
EC00413=798156,1112951
EC00414=798156,1112951
EC00415=798156,1112951
EC00416=798156,1112951
EC00417=798156,1112951
EC00418=798156,1112951
EC00419=798156,1112951
EC00420=798156,1112951
EC00421=798156,1112951
EC00422=798156,1112951
EC00423=798156,1112951
EC00424=798156,1112951
EC00425=798156,1112951
EC00426=798156,1112951
EC00427=798156,1112951
EC00428=798156,1112951
EC00429=798156,1112951
EC00430=798156,1112951
EC00431=798156,1112951
EC00432=798156,1112951
EC00433=798156,1112951
EC00434=798156,1112951
EC00435=798156,1112951
EC00436=798156,1112951
EC00437=798156,1112951
EC00438=798156,1112951
EC00439=798156,1112951
EC00440=798156,1112951
EC00441=798156,1112951
EC00442=798156,1112951
EC00443=798156,1112951
EC00444=798156,1112951
EC00445=798156,1112951
EC00446=798156,1112951
EC00447=798156,1112951
EC00448=798156,1112951
EC00449=798156,1112951
EC00450=798156,1112951
EC00451=798156,1112951
EC00452=798156,1112951
EC00453=798156,1112951
EC00454=798156,1112951
EC00455=798156,1112951
EC00456=798156,1112951
EC00457=798156,1112951
EC00458=798156,1112951
EC00459=798156,1112951
EC00460=798156,1112951
EC00461=798156,1112951
EC00462=798156,1112951
EC00463=798156,1112951
EC00464=798156,1112951
EC00465=798156,1112951
EC00466=798156,1112951
EC00467=798156,1112951
EC00468=798156,1112951
EC00469=798156,1112951
EC00470=798156,1112951
EC00471=798156,1112951
EC00472=798156,1112951
EC00473=798156,1112951
EC00474=798156,1112951
EC00475=798156,1112951
EC00476=798156,1112951
EC00477=798156,1112951
EC00478=798156,1112951
EC00479=798156,1112951
EC00480=798156,1112951
EC00481=798156,1112951
EC00482=798156,1112951
EC00483=798156,1112951
EC00484=798156,1112951
EC00485=798156,1112951
EC00486=798156,1112951
EC00487=798156,1112951
EC00488=798156,1112951
EC00489=798156,1112951
EC00490=798156,1112951
EC00491=798156,1112951
EC00492=798156,1112951
EC00493=798156,1112951
EC00494=798156,1112951
EC00495=798156,1112951
EC00496=798156,1112951
EC00497=798156,1112951
EC00498=798156,1112951
EC00499=798156,1112951
EC00500=798156,1112951
EC00501=798156,1112951
EC00502=798156,1112951
EC00503=798156,1112951
EC00504=798156,1112951
EC00505=798156,1112951
EC00506=798156,1112951
EC00507=798156,1112951
EC00508=798156,1112951
EC00509=798156,1112951
EC00510=798156,1112951
EC00511=798156,1112951
EC00512=798156,1112951
EC00513=798156,1112951
EC00514=798156,1112951
EC00515=798156,1112951
EC00516=798156,1112951
EC00517=798156,1112951
EC00518=798156,1112951
EC00519=798156,1112951
EC00520=798156,1112951
EC00521=798156,1112951
EC00522=798156,1112951
EC00523=798156,1112951
EC00524=798156,1112951
EC00525=798156,1112951
EC00526=798156,1112951
EC00527=798156,1112951
EC00528=798156,1112951
EC00529=798156,1112951
EC00530=798156,1112951
EC00531=798156,1112951
EC00532=798156,1112951
EC00533=798156,1112951
EC00534=798156,1112951
EC00535=798156,1112951
EC00536=798156,1112951
EC00537=798156,1112951
EC00538=798156,1112951
EC00539=798156,1112951
EC00540=798156,1112951
EC00541=798156,1112951
EC00542=798156,1112951
EC00543=798156,1112951
EC00544=798156,1112951
EC00545=798156,1112951
EC00546=798156,1112951
EC00547=798156,1112951
EC00548=798156,1112951
EC00549=798156,1112951
EC00550=798156,1112951
EC00551=798156,1112951
EC00552=798156,1112951
EC00553=798156,1112951
EC00554=798156,1112951
EC00555=798156,1112951
EC00556=798156,1112951
EC00557=798156,1112951
EC00558=798156,1112951
EC00559=798156,1112951
EC00560=798156,1112951
EC00561=798156,1112951
EC00562=798156,1112951
EC00563=798156,1112951
EC00564=798156,1112951
EC00565=798156,1112951
EC00566=798156,1112951
EC00567=798156,1112951
EC00568=798156,1112951
EC00569=798156,1112951
EC00570=798156,1112951
EC00571=798156,1112951
EC00572=798156,1112951
EC00573=798156,1112951
EC00574=798156,1112951
EC00575=798156,1112951
EC00576=798156,1112951
EC00577=798156,1112951
EC00578=798156,1112951
EC00579=798156,1112951
EC00580=798156,1112951
EC00581=798156,1112951
EC00582=798156,1112951
EC00583=798156,1112951
EC00584=798156,1112951
EC00585=798156,1112951
EC00586=798156,1112951
EC00587=798156,1112951
EC00588=798156,1112951
EC00589=798156,1112951
EC00590=798156,1112951
EC00591=798156,1112951
EC00592=798156,1112951
EC00593=798156,1112951
EC00594=798156,1112951
EC00595=798156,1112951
EC00596=798156,1112951
EC00597=798156,1112951
EC00598=798156,1112951
EC00599=798156,1112951
EC00600=798156,1112951
EC00601=798156,1112951
EC00602=798156,1112951
EC00603=798156,1112951
EC00604=798156,1112951
EC00605=798156,1112951
EC00606=798156,1112951
EC00607=798156,1112951
EC00608=798156,1112951
EC00609=798156,1112951
EC00610=798156,1112951
EC00611=798156,1112951
EC00612=798156,1112951
EC00613=798156,1112951
EC00614=798156,1112951
EC00615=798156,1112951
EC00616=798156,1112951
EC00617=798156,1112951
EC00618=798156,1112951
EC00619=798156,1112951
EC00620=798156,1112951
EC00621=798156,1112951
EC00622=798156,1112951
EC00623=798156,1112951
EC00624=798156,1112951
EC00625=798156,1112951
EC00626=798156,1112951
EC00627=798156,1112951
EC00628=798156,1112951
EC00629=798156,1112951
EC00630=798156,1112951
EC00631=798156,1112951
EC00632=798156,1112951
EC00633=798156,1112951
EC00634=798156,1112951
EC00635=798156,1112951
EC00636=798156,1112951
EC00637=798156,1112951
EC00638=798156,1112951
EC00639=798156,1112951
EC00640=798156,1112951
EC00641=798156,1112951
///POSTYPE BASE
///RECTAN
///RCONF 0,0,0,0,0,0,0,0,0,0,0,0,0,0,0,0,0,0,0,0,0,0,0,0
P00006=0.222,-3.123,-1.508,0.0000,0.0000,0.0000
P00021=-0.225,-6.128,-0.405,0.0000,0.0000,0.0000
P00022=0.222,-3.123,-1.508,0.0000,0.0000,0.0000
P00023=0.143,-0.036,0.682,0.0000,0.0000,0.0000
P00024=0.145,-0.552,1.326,0.0000,0.0000,0.0000
P00025=-2.003,0.006,0.728,0.0000,0.0000,0.0000
P00026=0.562,-0.002,-0.337,0.0000,0.0000,0.0000
P00027=-0.746,0.015,-9.096,0.0000,0.0000,0.0000
P00028=-2.237,-0.018,-7.702,0.0000,0.0000,0.0000
P00029=-2.156,-0.086,-4.681,0.0000,0.0000,0.0000
P00030=5.926,-4.294,-1.390,0.0000,0.0000,0.0000
P00031=1.853,-0.001,-1.549,0.0000,0.0000,0.0000
P00032=1.957,0.503,-7.217,0.0000,0.0000,0.0000
P00041=0.192,3.924,0.305,0.0000,0.0000,0.0000
P00042=-0.217,1.941,0.413,0.0000,0.0000,0.0000
P00043=-0.044,-1.937,1.197,0.0000,0.0000,0.0000
P00044=0.687,-2.322,1.156,0.0000,0.0000,0.0000
P00045=-0.068,-0.810,1.603,0.0000,0.0000,0.0000
//INST
///DATE 2024/01/09 18:53
///ATTR SC,RW
///GROUP1 RB1,BS1
///GROUP2 ST1
NOP
'r2_O57-69(2)(90,180)
'Down
'Path S1657
SSFTOF
MOVJ C00000 BC00000 VJ=100.00  +MOVJ EC00000 VJ=100.00
MOVL C00001 BC00001 V=100.0  +MOVJ EC00001 VJ=100.00
SMOVL C00002 BC00002 V=60.0  +MOVJ EC00002
SREFP 3 C00003 BC00003  +REFP EC00003
CALL JOB:SEARCH-R1-S1
SET P031 P006
SSFTON P031
SMOVL C00004 BC00004 V=60.0  +MOVJ EC00004
SMOVL C00005 BC00005 V=60.0  +MOVJ EC00005
SREFP 3 C00006 BC00006  +REFP EC00006
CALL JOB:SEARCH-R1-S1
SET P031 P006
SSFTON P031
SMOVL C00007 BC00007 V=60.0  +MOVJ EC00007
MOVL C00008 BC00008 V=400.0  +MOVJ EC00008 VJ=100.00
MOVL C00009 BC00009 V=1000.0  +MOVJ EC00009 VJ=100.00
'Path S1661
SSFTOF
MOVJ C00010 BC00010 VJ=100.00  +MOVJ EC00010 VJ=100.00
MOVL C00011 BC00011 V=100.0  +MOVJ EC00011 VJ=100.00
SMOVL C00012 BC00012 V=60.0  +MOVJ EC00012
SREFP 3 C00013 BC00013  +REFP EC00013
CALL JOB:SEARCH-R1-S1
SET P026 P006
SSFTON P026
SMOVL C00014 BC00014 V=60.0  +MOVJ EC00014
SMOVL C00015 BC00015 V=60.0  +MOVJ EC00015
SREFP 3 C00016 BC00016  +REFP EC00016
CALL JOB:SEARCH-R1-S1
SET P026 P006
SSFTON P026
SMOVL C00017 BC00017 V=60.0  +MOVJ EC00017
MOVL C00018 BC00018 V=400.0  +MOVJ EC00018 VJ=100.00
MOVL C00019 BC00019 V=1000.0  +MOVJ EC00019 VJ=100.00
'Path S1662
SSFTOF
MOVJ C00020 BC00020 VJ=100.00  +MOVJ EC00020 VJ=100.00
MOVL C00021 BC00021 V=100.0  +MOVJ EC00021 VJ=100.00
SMOVL C00022 BC00022 V=60.0  +MOVJ EC00022
SREFP 3 C00023 BC00023  +REFP EC00023
CALL JOB:SEARCH-R1-S1
SET P027 P006
SSFTON P027
SMOVL C00024 BC00024 V=60.0  +MOVJ EC00024
SMOVL C00025 BC00025 V=60.0  +MOVJ EC00025
SREFP 3 C00026 BC00026  +REFP EC00026
CALL JOB:SEARCH-R1-S1
SET P027 P006
SSFTON P027
SMOVL C00027 BC00027 V=60.0  +MOVJ EC00027
MOVL C00028 BC00028 V=400.0  +MOVJ EC00028 VJ=100.00
MOVL C00029 BC00029 V=1000.0  +MOVJ EC00029 VJ=100.00
MOVJ C00030 BC00030 VJ=100.00  +MOVJ EC00030 VJ=100.00
MOVJ C00031 BC00031 VJ=100.00  +MOVJ EC00031 VJ=100.00
'Path S1663
SSFTOF
MOVJ C00032 BC00032 VJ=100.00  +MOVJ EC00032 VJ=100.00
MOVL C00033 BC00033 V=100.0  +MOVJ EC00033 VJ=100.00
SMOVL C00034 BC00034 V=60.0  +MOVJ EC00034
SREFP 3 C00035 BC00035  +REFP EC00035
CALL JOB:SEARCH-R1-S1
SET P022 P006
SSFTON P022
SMOVL C00036 BC00036 V=60.0  +MOVJ EC00036
SMOVL C00037 BC00037 V=60.0  +MOVJ EC00037
SREFP 3 C00038 BC00038  +REFP EC00038
CALL JOB:SEARCH-R1-S1
SET P022 P006
SSFTON P022
SMOVL C00039 BC00039 V=60.0  +MOVJ EC00039
MOVL C00040 BC00040 V=400.0  +MOVJ EC00040 VJ=100.00
MOVL C00041 BC00041 V=1000.0  +MOVJ EC00041 VJ=100.00
MOVJ C00042 BC00042 VJ=100.00  +MOVJ EC00042 VJ=100.00
MOVJ C00043 BC00043 VJ=100.00  +MOVJ EC00043 VJ=100.00
MOVJ C00044 BC00044 VJ=100.00  +MOVJ EC00044 VJ=100.00
MOVJ C00045 BC00045 VJ=100.00  +MOVJ EC00045 VJ=100.00
'Path S1658
SSFTOF
MOVJ C00046 BC00046 VJ=100.00  +MOVJ EC00046 VJ=100.00
MOVL C00047 BC00047 V=100.0  +MOVJ EC00047 VJ=100.00
SMOVL C00048 BC00048 V=60.0  +MOVJ EC00048
SREFP 3 C00049 BC00049  +REFP EC00049
CALL JOB:SEARCH-R1-S1
SET P028 P006
SSFTON P028
SMOVL C00050 BC00050 V=60.0  +MOVJ EC00050
SMOVL C00051 BC00051 V=60.0  +MOVJ EC00051
SREFP 3 C00052 BC00052  +REFP EC00052
CALL JOB:SEARCH-R1-S1
SET P028 P006
SSFTON P028
SMOVL C00053 BC00053 V=60.0  +MOVJ EC00053
MOVL C00054 BC00054 V=400.0  +MOVJ EC00054 VJ=100.00
MOVL C00055 BC00055 V=1000.0  +MOVJ EC00055 VJ=100.00
'Path S1659
SSFTOF
MOVJ C00056 BC00056 VJ=100.00  +MOVJ EC00056 VJ=100.00
MOVL C00057 BC00057 V=100.0  +MOVJ EC00057 VJ=100.00
SMOVL C00058 BC00058 V=60.0  +MOVJ EC00058
SREFP 3 C00059 BC00059  +REFP EC00059
CALL JOB:SEARCH-R1-S1
SET P029 P006
SSFTON P029
SMOVL C00060 BC00060 V=60.0  +MOVJ EC00060
SMOVL C00061 BC00061 V=60.0  +MOVJ EC00061
SREFP 3 C00062 BC00062  +REFP EC00062
CALL JOB:SEARCH-R1-S1
SET P029 P006
SSFTON P029
SMOVL C00063 BC00063 V=60.0  +MOVJ EC00063
MOVL C00064 BC00064 V=400.0  +MOVJ EC00064 VJ=100.00
MOVL C00065 BC00065 V=1000.0  +MOVJ EC00065 VJ=100.00
'Path S1660
SSFTOF
MOVJ C00066 BC00066 VJ=100.00  +MOVJ EC00066 VJ=100.00
MOVL C00067 BC00067 V=100.0  +MOVJ EC00067 VJ=100.00
SMOVL C00068 BC00068 V=60.0  +MOVJ EC00068
SREFP 3 C00069 BC00069  +REFP EC00069
CALL JOB:SEARCH-R1-S1
SET P030 P006
SSFTON P030
SMOVL C00070 BC00070 V=60.0  +MOVJ EC00070
SMOVL C00071 BC00071 V=60.0  +MOVJ EC00071
SREFP 3 C00072 BC00072  +REFP EC00072
CALL JOB:SEARCH-R1-S1
SET P030 P006
SSFTON P030
SMOVL C00073 BC00073 V=60.0  +MOVJ EC00073
MOVL C00074 BC00074 V=400.0  +MOVJ EC00074 VJ=100.00
MOVL C00075 BC00075 V=1000.0  +MOVJ EC00075 VJ=100.00
'Path S1664
SSFTOF
MOVJ C00076 BC00076 VJ=100.00  +MOVJ EC00076 VJ=100.00
MOVL C00077 BC00077 V=400.0  +MOVJ EC00077 VJ=100.00
SMOVL C00078 BC00078 V=60.0  +MOVJ EC00078
SREFP 3 C00079 BC00079  +REFP EC00079
CALL JOB:SEARCH-R1-S1
SET P023 P006
SSFTON P023
SMOVL C00080 BC00080 V=60.0  +MOVJ EC00080
SMOVL C00081 BC00081 V=60.0  +MOVJ EC00081
SREFP 3 C00082 BC00082  +REFP EC00082
CALL JOB:SEARCH-R1-S1
SET P023 P006
SSFTON P023
SMOVL C00083 BC00083 V=60.0  +MOVJ EC00083
SMOVL C00084 BC00084 V=60.0  +MOVJ EC00084
SREFP 3 C00085 BC00085  +REFP EC00085
CALL JOB:SEARCH-R1-S1
SET P023 P006
SSFTON P023
SMOVL C00086 BC00086 V=60.0  +MOVJ EC00086
MOVL C00087 BC00087 V=400.0  +MOVJ EC00087 VJ=100.00
MOVL C00088 BC00088 V=1000.0  +MOVJ EC00088 VJ=100.00
'Path S1665
SSFTOF
MOVJ C00089 BC00089 VJ=100.00  +MOVJ EC00089 VJ=100.00
MOVL C00090 BC00090 V=100.0  +MOVJ EC00090 VJ=100.00
SMOVL C00091 BC00091 V=60.0  +MOVJ EC00091
SREFP 3 C00092 BC00092  +REFP EC00092
CALL JOB:SEARCH-R1-S1
SET P024 P006
SSFTON P024
SMOVL C00093 BC00093 V=60.0  +MOVJ EC00093
SMOVL C00094 BC00094 V=60.0  +MOVJ EC00094
SREFP 3 C00095 BC00095  +REFP EC00095
CALL JOB:SEARCH-R1-S1
SET P024 P006
SSFTON P024
SMOVL C00096 BC00096 V=60.0  +MOVJ EC00096
SMOVL C00097 BC00097 V=60.0  +MOVJ EC00097
SREFP 3 C00098 BC00098  +REFP EC00098
CALL JOB:SEARCH-R1-S1
SET P024 P006
SSFTON P024
SMOVL C00099 BC00099 V=60.0  +MOVJ EC00099
MOVL C00100 BC00100 V=400.0  +MOVJ EC00100 VJ=100.00
MOVL C00101 BC00101 V=1000.0  +MOVJ EC00101 VJ=100.00
MOVJ C00102 BC00102 VJ=100.00  +MOVJ EC00102 VJ=100.00
'Path S1666
SSFTOF
MOVJ C00103 BC00103 VJ=100.00  +MOVJ EC00103 VJ=100.00
MOVL C00104 BC00104 V=400.0  +MOVJ EC00104 VJ=100.00
SMOVL C00105 BC00105 V=60.0  +MOVJ EC00105
SREFP 3 C00106 BC00106  +REFP EC00106
CALL JOB:SEARCH-R1-S1
SET P025 P006
SSFTON P025
SMOVL C00107 BC00107 V=60.0  +MOVJ EC00107
SMOVL C00108 BC00108 V=60.0  +MOVJ EC00108
SREFP 3 C00109 BC00109  +REFP EC00109
CALL JOB:SEARCH-R1-S1
SET P025 P006
SSFTON P025
SMOVL C00110 BC00110 V=60.0  +MOVJ EC00110
SMOVL C00111 BC00111 V=60.0  +MOVJ EC00111
SREFP 3 C00112 BC00112  +REFP EC00112
CALL JOB:SEARCH-R1-S1
SET P025 P006
SSFTON P025
SMOVL C00113 BC00113 V=60.0  +MOVJ EC00113
MOVL C00114 BC00114 V=400.0  +MOVJ EC00114 VJ=100.00
MOVL C00115 BC00115 V=1000.0  +MOVJ EC00115 VJ=100.00
MOVJ C00116 BC00116 VJ=100.00  +MOVJ EC00116 VJ=100.00
MOVJ C00117 BC00117 VJ=100.00  +MOVJ EC00117 VJ=100.00
'Path S1667
SSFTOF
MOVJ C00118 BC00118 VJ=100.00  +MOVJ EC00118 VJ=100.00
MOVL C00119 BC00119 V=400.0  +MOVJ EC00119 VJ=100.00
SMOVL C00120 BC00120 V=60.0  +MOVJ EC00120
SREFP 3 C00121 BC00121  +REFP EC00121
CALL JOB:SEARCH-R1-S1
SET P021 P006
SSFTON P021
SMOVL C00122 BC00122 V=60.0  +MOVJ EC00122
SMOVL C00123 BC00123 V=60.0  +MOVJ EC00123
SREFP 3 C00124 BC00124  +REFP EC00124
CALL JOB:SEARCH-R1-S1
SET P021 P006
SSFTON P021
SMOVL C00125 BC00125 V=60.0  +MOVJ EC00125
SMOVL C00126 BC00126 V=60.0  +MOVJ EC00126
SREFP 3 C00127 BC00127  +REFP EC00127
CALL JOB:SEARCH-R1-S1
SET P021 P006
SSFTON P021
SMOVL C00128 BC00128 V=60.0  +MOVJ EC00128
MOVL C00129 BC00129 V=400.0  +MOVJ EC00129 VJ=100.00
MOVL C00130 BC00130 V=1000.0  +MOVJ EC00130 VJ=100.00
MOVJ C00131 BC00131 VJ=100.00  +MOVJ EC00131 VJ=100.00
'Path S2042
SSFTOF
MOVJ C00132 BC00132 VJ=100.00  +MOVJ EC00132 VJ=100.00
MOVL C00133 BC00133 V=400.0  +MOVJ EC00133 VJ=100.00
SMOVL C00134 BC00134 V=60.0  +MOVJ EC00134
SREFP 3 C00135 BC00135  +REFP EC00135
CALL JOB:SEARCH-R1-S1
SET P032 P006
SSFTON P032
SMOVL C00136 BC00136 V=60.0  +MOVJ EC00136
SMOVL C00137 BC00137 V=60.0  +MOVJ EC00137
SREFP 3 C00138 BC00138  +REFP EC00138
CALL JOB:SEARCH-R1-S1
SET P032 P006
SSFTON P032
SMOVL C00139 BC00139 V=60.0  +MOVJ EC00139
MOVL C00140 BC00140 V=400.0  +MOVJ EC00140 VJ=100.00
MOVL C00141 BC00141 V=1000.0  +MOVJ EC00141 VJ=100.00
MOVJ C00142 BC00142 VJ=100.00  +MOVJ EC00142 VJ=100.00
MOVJ C00143 BC00143 VJ=100.00  +MOVJ EC00143 VJ=100.00
MOVJ C00144 BC00144 VJ=100.00  +MOVJ EC00144 VJ=100.00
MOVJ C00145 BC00145 VJ=100.00  +MOVJ EC00145 VJ=100.00
'Up
'Path S1190
SSFTOF
MOVJ C00146 BC00146 VJ=100.00  +MOVJ EC00146 VJ=100.00
MOVL C00147 BC00147 V=400.0  +MOVJ EC00147 VJ=100.00
SMOVL C00148 BC00148 V=60.0  +MOVJ EC00148
SREFP 3 C00149 BC00149  +REFP EC00149
CALL JOB:SEARCH-R1-S1
SET P045 P006
SSFTON P045
SMOVL C00150 BC00150 V=60.0  +MOVJ EC00150
SMOVL C00151 BC00151 V=60.0  +MOVJ EC00151
SREFP 3 C00152 BC00152  +REFP EC00152
CALL JOB:SEARCH-R1-S1
SET P045 P006
SSFTON P045
SMOVL C00153 BC00153 V=60.0  +MOVJ EC00153
MOVL C00154 BC00154 V=400.0  +MOVJ EC00154 VJ=100.00
MOVL C00155 BC00155 V=1000.0  +MOVJ EC00155 VJ=100.00
'Path S1972
SSFTOF
MOVJ C00156 BC00156 VJ=100.00  +MOVJ EC00156 VJ=100.00
MOVL C00157 BC00157 V=400.0  +MOVJ EC00157 VJ=100.00
SMOVL C00158 BC00158 V=60.0  +MOVJ EC00158
SREFP 3 C00159 BC00159  +REFP EC00159
CALL JOB:SEARCH-R1-S1
SET P044 P006
SSFTON P044
SMOVL C00160 BC00160 V=60.0  +MOVJ EC00160
SMOVL C00161 BC00161 V=60.0  +MOVJ EC00161
SREFP 3 C00162 BC00162  +REFP EC00162
CALL JOB:SEARCH-R1-S1
SET P044 P006
SSFTON P044
SMOVL C00163 BC00163 V=60.0  +MOVJ EC00163
MOVL C00164 BC00164 V=400.0  +MOVJ EC00164 VJ=100.00
MOVL C00165 BC00165 V=1000.0  +MOVJ EC00165 VJ=100.00
'Path S1189
SSFTOF
MOVJ C00166 BC00166 VJ=100.00  +MOVJ EC00166 VJ=100.00
MOVL C00167 BC00167 V=400.0  +MOVJ EC00167 VJ=100.00
SMOVL C00168 BC00168 V=60.0  +MOVJ EC00168
SREFP 3 C00169 BC00169  +REFP EC00169
CALL JOB:SEARCH-R1-S1
SET P043 P006
SSFTON P043
SMOVL C00170 BC00170 V=60.0  +MOVJ EC00170
SMOVL C00171 BC00171 V=60.0  +MOVJ EC00171
SREFP 3 C00172 BC00172  +REFP EC00172
CALL JOB:SEARCH-R1-S1
SET P043 P006
SSFTON P043
SMOVL C00173 BC00173 V=60.0  +MOVJ EC00173
MOVL C00174 BC00174 V=400.0  +MOVJ EC00174 VJ=100.00
MOVL C00175 BC00175 V=1000.0  +MOVJ EC00175 VJ=100.00
MOVJ C00176 BC00176 VJ=100.00  +MOVJ EC00176 VJ=100.00
'Path S1188
SSFTOF
MOVJ C00177 BC00177 VJ=100.00  +MOVJ EC00177 VJ=100.00
MOVL C00178 BC00178 V=400.0  +MOVJ EC00178 VJ=100.00
SMOVL C00179 BC00179 V=60.0  +MOVJ EC00179
SREFP 3 C00180 BC00180  +REFP EC00180
CALL JOB:SEARCH-R1-S1
SET P042 P006
SSFTON P042
SMOVL C00181 BC00181 V=60.0  +MOVJ EC00181
SMOVL C00182 BC00182 V=60.0  +MOVJ EC00182
SREFP 3 C00183 BC00183  +REFP EC00183
CALL JOB:SEARCH-R1-S1
SET P042 P006
SSFTON P042
SMOVL C00184 BC00184 V=60.0  +MOVJ EC00184
SMOVL C00185 BC00185 V=60.0  +MOVJ EC00185
SREFP 3 C00186 BC00186  +REFP EC00186
CALL JOB:SEARCH-R1-S1
SET P042 P006
SSFTON P042
SMOVL C00187 BC00187 V=60.0  +MOVJ EC00187
MOVL C00188 BC00188 V=400.0  +MOVJ EC00188 VJ=100.00
MOVL C00189 BC00189 V=1000.0  +MOVJ EC00189 VJ=100.00
'Path S1187
SSFTOF
MOVJ C00190 BC00190 VJ=100.00  +MOVJ EC00190 VJ=100.00
MOVL C00191 BC00191 V=400.0  +MOVJ EC00191 VJ=100.00
SMOVL C00192 BC00192 V=60.0  +MOVJ EC00192
SREFP 3 C00193 BC00193  +REFP EC00193
CALL JOB:SEARCH-R1-S1
SET P041 P006
SSFTON P041
SMOVL C00194 BC00194 V=60.0  +MOVJ EC00194
SMOVL C00195 BC00195 V=60.0  +MOVJ EC00195
SREFP 3 C00196 BC00196  +REFP EC00196
CALL JOB:SEARCH-R1-S1
SET P041 P006
SSFTON P041
SMOVL C00197 BC00197 V=60.0  +MOVJ EC00197
SMOVL C00198 BC00198 V=60.0  +MOVJ EC00198
SREFP 3 C00199 BC00199  +REFP EC00199
CALL JOB:SEARCH-R1-S1
SET P041 P006
SSFTON P041
SMOVL C00200 BC00200 V=60.0  +MOVJ EC00200
MOVL C00201 BC00201 V=400.0  +MOVJ EC00201 VJ=100.00
MOVL C00202 BC00202 V=1000.0  +MOVJ EC00202 VJ=100.00
'Path W1181
SSFTOF
SSFTON P041
MOVJ C00203 BC00203 VJ=100.00  +MOVJ EC00203 VJ=100.00
SMOVL C00204 BC00204 V=400.0  +MOVJ EC00204
SMOVL C00205 BC00205 V=100.0 PL=0  +MOVJ EC00205
SREFP 1 C00206 BC00206  +REFP EC00206
SREFP 2 C00207 BC00207  +REFP EC00207
MACRO1 MJ#(0) ARGF0
ARCON
SMOVL C00208 BC00208 V=10.0  +MOVJ EC00208
SMOVL C00209 BC00209 V=10.0  +MOVJ EC00209
SMOVL C00210 BC00210 V=10.0  +MOVJ EC00210
ARCOF
SMOVL C00211 BC00211 V=400.0  +MOVJ EC00211
SMOVL C00212 BC00212 V=1000.0  +MOVJ EC00212
SSFTOF
MOVJ C00213 BC00213 VJ=100.00  +MOVJ EC00213 VJ=100.00
'Path W1182
SSFTOF
SSFTON P042
MOVJ C00214 BC00214 VJ=100.00  +MOVJ EC00214 VJ=100.00
SMOVL C00215 BC00215 V=400.0  +MOVJ EC00215
SMOVL C00216 BC00216 V=100.0 PL=0  +MOVJ EC00216
SREFP 1 C00217 BC00217  +REFP EC00217
SREFP 2 C00218 BC00218  +REFP EC00218
MACRO1 MJ#(0) ARGF0
ARCON
SMOVL C00219 BC00219 V=10.0  +MOVJ EC00219
SMOVL C00220 BC00220 V=10.0  +MOVJ EC00220
SMOVL C00221 BC00221 V=10.0  +MOVJ EC00221
ARCOF
SMOVL C00222 BC00222 V=400.0  +MOVJ EC00222
SMOVL C00223 BC00223 V=1000.0  +MOVJ EC00223
SSFTOF
MOVJ C00224 BC00224 VJ=100.00  +MOVJ EC00224 VJ=100.00
'Path W1192
SSFTOF
SSFTON P045
MOVJ C00225 BC00225 VJ=100.00  +MOVJ EC00225 VJ=100.00
SMOVL C00226 BC00226 V=400.0  +MOVJ EC00226
SMOVL C00227 BC00227 V=100.0 PL=0  +MOVJ EC00227
SREFP 1 C00228 BC00228  +REFP EC00228
SREFP 2 C00229 BC00229  +REFP EC00229
MACRO1 MJ#(0) ARGF0
ARCON
SMOVL C00230 BC00230 V=10.0  +MOVJ EC00230
SMOVL C00231 BC00231 V=10.0  +MOVJ EC00231
SMOVL C00232 BC00232 V=10.0  +MOVJ EC00232
SMOVL C00233 BC00233 V=10.0  +MOVJ EC00233
SMOVL C00234 BC00234 V=10.0  +MOVJ EC00234
SMOVL C00235 BC00235 V=10.0  +MOVJ EC00235
SMOVL C00236 BC00236 V=10.0  +MOVJ EC00236
SMOVL C00237 BC00237 V=10.0  +MOVJ EC00237
SMOVL C00238 BC00238 V=10.0  +MOVJ EC00238
SMOVL C00239 BC00239 V=10.0  +MOVJ EC00239
SMOVL C00240 BC00240 V=10.0  +MOVJ EC00240
SMOVL C00241 BC00241 V=10.0  +MOVJ EC00241
SMOVL C00242 BC00242 V=10.0  +MOVJ EC00242
SMOVL C00243 BC00243 V=10.0  +MOVJ EC00243
SMOVL C00244 BC00244 V=10.0  +MOVJ EC00244
SMOVL C00245 BC00245 V=10.0  +MOVJ EC00245
SMOVL C00246 BC00246 V=10.0  +MOVJ EC00246
SMOVL C00247 BC00247 V=10.0  +MOVJ EC00247
SMOVL C00248 BC00248 V=10.0  +MOVJ EC00248
SMOVL C00249 BC00249 V=10.0  +MOVJ EC00249
SMOVL C00250 BC00250 V=10.0  +MOVJ EC00250
SMOVL C00251 BC00251 V=10.0  +MOVJ EC00251
SMOVL C00252 BC00252 V=10.0  +MOVJ EC00252
SMOVL C00253 BC00253 V=10.0  +MOVJ EC00253
SMOVL C00254 BC00254 V=10.0  +MOVJ EC00254
SMOVL C00255 BC00255 V=10.0  +MOVJ EC00255
SMOVL C00256 BC00256 V=10.0  +MOVJ EC00256
ARCOF
SMOVL C00257 BC00257 V=400.0  +MOVJ EC00257
SMOVL C00258 BC00258 V=1000.0  +MOVJ EC00258
SSFTOF
'Path W1184
SSFTOF
SSFTON P044
MOVJ C00259 BC00259 VJ=100.00  +MOVJ EC00259 VJ=100.00
SMOVL C00260 BC00260 V=400.0  +MOVJ EC00260
SMOVL C00261 BC00261 V=100.0 PL=0  +MOVJ EC00261
SREFP 1 C00262 BC00262  +REFP EC00262
SREFP 2 C00263 BC00263  +REFP EC00263
MACRO1 MJ#(0) ARGF0
ARCON
SMOVL C00264 BC00264 V=10.0  +MOVJ EC00264
SMOVL C00265 BC00265 V=10.0  +MOVJ EC00265
SMOVL C00266 BC00266 V=10.0  +MOVJ EC00266
ARCOF
SMOVL C00267 BC00267 V=400.0  +MOVJ EC00267
SMOVL C00268 BC00268 V=1000.0  +MOVJ EC00268
SSFTOF
MOVJ C00269 BC00269 VJ=100.00  +MOVJ EC00269 VJ=100.00
'Path W1185
SSFTOF
SSFTON P043
MOVJ C00270 BC00270 VJ=100.00  +MOVJ EC00270 VJ=100.00
SMOVL C00271 BC00271 V=400.0  +MOVJ EC00271
SMOVL C00272 BC00272 V=100.0 PL=0  +MOVJ EC00272
SREFP 1 C00273 BC00273  +REFP EC00273
SREFP 2 C00274 BC00274  +REFP EC00274
MACRO1 MJ#(0) ARGF0
ARCON
SMOVL C00275 BC00275 V=10.0  +MOVJ EC00275
SMOVL C00276 BC00276 V=10.0  +MOVJ EC00276
SMOVL C00277 BC00277 V=10.0  +MOVJ EC00277
ARCOF
SMOVL C00278 BC00278 V=400.0  +MOVJ EC00278
SMOVL C00279 BC00279 V=1000.0  +MOVJ EC00279
SSFTOF
MOVJ C00280 BC00280 VJ=100.00  +MOVJ EC00280 VJ=100.00
MOVJ C00281 BC00281 VJ=100.00  +MOVJ EC00281 VJ=100.00
MOVJ C00282 BC00282 VJ=100.00  +MOVJ EC00282 VJ=100.00
MOVJ C00283 BC00283 VJ=100.00  +MOVJ EC00283 VJ=100.00
'Down
'Path W1668
SSFTOF
SSFTON P021
MOVJ C00284 BC00284 VJ=100.00  +MOVJ EC00284 VJ=100.00
SMOVL C00285 BC00285 V=400.0  +MOVJ EC00285
SMOVL C00286 BC00286 V=100.0 PL=0  +MOVJ EC00286
SREFP 1 C00287 BC00287  +REFP EC00287
SREFP 2 C00288 BC00288  +REFP EC00288
MACRO1 MJ#(0) ARGF0
ARCON
SMOVL C00289 BC00289 V=10.0  +MOVJ EC00289
SMOVL C00290 BC00290 V=10.0  +MOVJ EC00290
SMOVL C00291 BC00291 V=10.0  +MOVJ EC00291
SMOVL C00292 BC00292 V=10.0  +MOVJ EC00292
SMOVL C00293 BC00293 V=10.0  +MOVJ EC00293
SMOVL C00294 BC00294 V=10.0  +MOVJ EC00294
SMOVL C00295 BC00295 V=10.0  +MOVJ EC00295
SMOVL C00296 BC00296 V=10.0  +MOVJ EC00296
SMOVL C00297 BC00297 V=10.0  +MOVJ EC00297
SMOVL C00298 BC00298 V=10.0  +MOVJ EC00298
ARCOF
SMOVL C00299 BC00299 V=400.0  +MOVJ EC00299
SMOVL C00300 BC00300 V=1000.0  +MOVJ EC00300
SSFTOF
MOVJ C00301 BC00301 VJ=100.00  +MOVJ EC00301 VJ=100.00
MOVJ C00302 BC00302 VJ=100.00  +MOVJ EC00302 VJ=100.00
'Path W1669
SSFTOF
SSFTON P032
MOVJ C00303 BC00303 VJ=100.00  +MOVJ EC00303 VJ=100.00
SMOVL C00304 BC00304 V=100.0  +MOVJ EC00304
SMOVL C00305 BC00305 V=100.0 PL=0  +MOVJ EC00305
SREFP 1 C00306 BC00306  +REFP EC00306
SREFP 2 C00307 BC00307  +REFP EC00307
MACRO1 MJ#(0) ARGF0
ARCON
SMOVL C00308 BC00308 V=10.0  +MOVJ EC00308
SMOVL C00309 BC00309 V=10.0  +MOVJ EC00309
SMOVL C00310 BC00310 V=10.0  +MOVJ EC00310
SMOVL C00311 BC00311 V=10.0  +MOVJ EC00311
SMOVL C00312 BC00312 V=10.0  +MOVJ EC00312
SMOVL C00313 BC00313 V=10.0  +MOVJ EC00313
SMOVL C00314 BC00314 V=10.0  +MOVJ EC00314
SMOVL C00315 BC00315 V=10.0  +MOVJ EC00315
SMOVL C00316 BC00316 V=10.0  +MOVJ EC00316
SMOVL C00317 BC00317 V=10.0  +MOVJ EC00317
SMOVL C00318 BC00318 V=10.0  +MOVJ EC00318
SMOVL C00319 BC00319 V=10.0  +MOVJ EC00319
ARCOF
SMOVL C00320 BC00320 V=400.0  +MOVJ EC00320
SMOVL C00321 BC00321 V=1000.0  +MOVJ EC00321
SSFTOF
MOVJ C00322 BC00322 VJ=100.00  +MOVJ EC00322 VJ=100.00
'
MOVJ C00323 BC00323 VJ=100.00  +MOVJ EC00323 VJ=100.00
MOVJ C00324 BC00324 VJ=100.00  +MOVJ EC00324 VJ=100.00
'Path W1670
SSFTOF
SSFTON P022
MOVJ C00325 BC00325 VJ=100.00  +MOVJ EC00325 VJ=100.00
SMOVL C00326 BC00326 V=100.0  +MOVJ EC00326
SMOVL C00327 BC00327 V=100.0 PL=0  +MOVJ EC00327
SREFP 1 C00328 BC00328  +REFP EC00328
SREFP 2 C00329 BC00329  +REFP EC00329
MACRO1 MJ#(0) ARGF0
ARCON
SMOVL C00330 BC00330 V=10.0  +MOVJ EC00330
SMOVL C00331 BC00331 V=10.0  +MOVJ EC00331
SMOVL C00332 BC00332 V=10.0  +MOVJ EC00332
SMOVL C00333 BC00333 V=10.0  +MOVJ EC00333
SMOVL C00334 BC00334 V=10.0  +MOVJ EC00334
SMOVL C00335 BC00335 V=10.0  +MOVJ EC00335
SMOVL C00336 BC00336 V=10.0  +MOVJ EC00336
ARCOF
SMOVL C00337 BC00337 V=400.0  +MOVJ EC00337
SMOVL C00338 BC00338 V=1000.0  +MOVJ EC00338
SSFTOF
'Path W1671
SSFTOF
SSFTON P022
MOVJ C00339 BC00339 VJ=100.00  +MOVJ EC00339 VJ=100.00
SMOVL C00340 BC00340 V=100.0  +MOVJ EC00340
SMOVL C00341 BC00341 V=100.0 PL=0  +MOVJ EC00341
SREFP 1 C00342 BC00342  +REFP EC00342
SREFP 2 C00343 BC00343  +REFP EC00343
MACRO1 MJ#(0) ARGF0
ARCON
SMOVL C00344 BC00344 V=10.0  +MOVJ EC00344
SMOVL C00345 BC00345 V=10.0  +MOVJ EC00345
SMOVL C00346 BC00346 V=10.0  +MOVJ EC00346
ARCOF
SMOVL C00347 BC00347 V=400.0  +MOVJ EC00347
SMOVL C00348 BC00348 V=1000.0  +MOVJ EC00348
SSFTOF
MOVJ C00349 BC00349 VJ=100.00  +MOVJ EC00349 VJ=100.00
MOVJ C00350 BC00350 VJ=100.00  +MOVJ EC00350 VJ=100.00
MOVJ C00351 BC00351 VJ=100.00  +MOVJ EC00351 VJ=100.00
'
MOVJ C00352 BC00352 VJ=100.00  +MOVJ EC00352 VJ=100.00
MOVJ C00353 BC00353 VJ=100.00  +MOVJ EC00353 VJ=100.00
'Path W1673
SSFTOF
SSFTON P023
MOVJ C00354 BC00354 VJ=100.00  +MOVJ EC00354 VJ=100.00
SMOVL C00355 BC00355 V=100.0  +MOVJ EC00355
SMOVL C00356 BC00356 V=100.0 PL=0  +MOVJ EC00356
SREFP 1 C00357 BC00357  +REFP EC00357
SREFP 2 C00358 BC00358  +REFP EC00358
MACRO1 MJ#(0) ARGF0
ARCON
SMOVL C00359 BC00359 V=10.0  +MOVJ EC00359
SMOVL C00360 BC00360 V=10.0  +MOVJ EC00360
SMOVL C00361 BC00361 V=10.0  +MOVJ EC00361
ARCOF
SMOVL C00362 BC00362 V=400.0  +MOVJ EC00362
SMOVL C00363 BC00363 V=1000.0  +MOVJ EC00363
SSFTOF
'Path W1674
SSFTOF
SSFTON P023
MOVJ C00364 BC00364 VJ=100.00  +MOVJ EC00364 VJ=100.00
SMOVL C00365 BC00365 V=100.0  +MOVJ EC00365
SMOVL C00366 BC00366 V=100.0 PL=0  +MOVJ EC00366
SREFP 1 C00367 BC00367  +REFP EC00367
SREFP 2 C00368 BC00368  +REFP EC00368
MACRO1 MJ#(0) ARGF0
ARCON
SMOVL C00369 BC00369 V=10.0  +MOVJ EC00369
SMOVL C00370 BC00370 V=10.0  +MOVJ EC00370
SMOVL C00371 BC00371 V=10.0  +MOVJ EC00371
ARCOF
SMOVL C00372 BC00372 V=400.0  +MOVJ EC00372
SMOVL C00373 BC00373 V=1000.0  +MOVJ EC00373
SSFTOF
'Path W1675
SSFTOF
SSFTON P023
MOVJ C00374 BC00374 VJ=100.00  +MOVJ EC00374 VJ=100.00
SMOVL C00375 BC00375 V=100.0  +MOVJ EC00375
SMOVL C00376 BC00376 V=100.0 PL=0  +MOVJ EC00376
SREFP 1 C00377 BC00377  +REFP EC00377
SREFP 2 C00378 BC00378  +REFP EC00378
MACRO1 MJ#(0) ARGF0
ARCON
SMOVL C00379 BC00379 V=10.0  +MOVJ EC00379
ARCOF
SMOVL C00380 BC00380 V=400.0  +MOVJ EC00380
SMOVL C00381 BC00381 V=1000.0  +MOVJ EC00381
SSFTOF
'
'Path W1676
SSFTOF
SSFTON P024
MOVJ C00382 BC00382 VJ=100.00  +MOVJ EC00382 VJ=100.00
SMOVL C00383 BC00383 V=100.0  +MOVJ EC00383
SMOVL C00384 BC00384 V=100.0 PL=0  +MOVJ EC00384
SREFP 1 C00385 BC00385  +REFP EC00385
SREFP 2 C00386 BC00386  +REFP EC00386
MACRO1 MJ#(0) ARGF0
ARCON
SMOVL C00387 BC00387 V=10.0  +MOVJ EC00387
SMOVL C00388 BC00388 V=10.0  +MOVJ EC00388
SMOVL C00389 BC00389 V=10.0  +MOVJ EC00389
ARCOF
SMOVL C00390 BC00390 V=400.0  +MOVJ EC00390
SMOVL C00391 BC00391 V=1000.0  +MOVJ EC00391
SSFTOF
MOVJ C00392 BC00392 VJ=100.00  +MOVJ EC00392 VJ=100.00
'Path W1677
SSFTOF
SSFTON P024
MOVJ C00393 BC00393 VJ=100.00  +MOVJ EC00393 VJ=100.00
SMOVL C00394 BC00394 V=100.0  +MOVJ EC00394
SMOVL C00395 BC00395 V=100.0 PL=0  +MOVJ EC00395
SREFP 1 C00396 BC00396  +REFP EC00396
SREFP 2 C00397 BC00397  +REFP EC00397
MACRO1 MJ#(0) ARGF0
ARCON
SMOVL C00398 BC00398 V=10.0  +MOVJ EC00398
SMOVL C00399 BC00399 V=10.0  +MOVJ EC00399
SMOVL C00400 BC00400 V=10.0  +MOVJ EC00400
ARCOF
SMOVL C00401 BC00401 V=400.0  +MOVJ EC00401
SMOVL C00402 BC00402 V=1000.0  +MOVJ EC00402
SSFTOF
'Path W1678
SSFTOF
SSFTON P024
MOVJ C00403 BC00403 VJ=100.00  +MOVJ EC00403 VJ=100.00
SMOVL C00404 BC00404 V=100.0  +MOVJ EC00404
SMOVL C00405 BC00405 V=100.0 PL=0  +MOVJ EC00405
SREFP 1 C00406 BC00406  +REFP EC00406
SREFP 2 C00407 BC00407  +REFP EC00407
MACRO1 MJ#(0) ARGF0
ARCON
SMOVL C00408 BC00408 V=10.0  +MOVJ EC00408
ARCOF
SMOVL C00409 BC00409 V=400.0  +MOVJ EC00409
SMOVL C00410 BC00410 V=1000.0  +MOVJ EC00410
SSFTOF
'
'Path W1680
SSFTOF
SSFTON P025
MOVJ C00411 BC00411 VJ=100.00  +MOVJ EC00411 VJ=100.00
SMOVL C00412 BC00412 V=100.0  +MOVJ EC00412
SMOVL C00413 BC00413 V=100.0 PL=0  +MOVJ EC00413
SREFP 1 C00414 BC00414  +REFP EC00414
SREFP 2 C00415 BC00415  +REFP EC00415
MACRO1 MJ#(0) ARGF0
ARCON
SMOVL C00416 BC00416 V=10.0  +MOVJ EC00416
SMOVL C00417 BC00417 V=10.0  +MOVJ EC00417
SMOVL C00418 BC00418 V=10.0  +MOVJ EC00418
ARCOF
SMOVL C00419 BC00419 V=400.0  +MOVJ EC00419
SMOVL C00420 BC00420 V=1000.0  +MOVJ EC00420
SSFTOF
MOVJ C00421 BC00421 VJ=100.00  +MOVJ EC00421 VJ=100.00
MOVJ C00422 BC00422 VJ=100.00  +MOVJ EC00422 VJ=100.00
MOVJ C00423 BC00423 VJ=100.00  +MOVJ EC00423 VJ=100.00
MOVJ C00424 BC00424 VJ=100.00  +MOVJ EC00424 VJ=100.00
MOVJ C00425 BC00425 VJ=100.00  +MOVJ EC00425 VJ=100.00
'Path W1679
SSFTOF
SSFTON P025
MOVJ C00426 BC00426 VJ=100.00  +MOVJ EC00426 VJ=100.00
SMOVL C00427 BC00427 V=100.0 PL=0  +MOVJ EC00427
SREFP 1 C00428 BC00428  +REFP EC00428
SREFP 2 C00429 BC00429  +REFP EC00429
MACRO1 MJ#(0) ARGF0
ARCON
SMOVL C00430 BC00430 V=10.0  +MOVJ EC00430
SMOVL C00431 BC00431 V=10.0  +MOVJ EC00431
SMOVL C00432 BC00432 V=10.0  +MOVJ EC00432
ARCOF
SMOVL C00433 BC00433 V=400.0  +MOVJ EC00433
SMOVL C00434 BC00434 V=1000.0  +MOVJ EC00434
SSFTOF
'Path W1681
SSFTOF
SSFTON P025
MOVJ C00435 BC00435 VJ=100.00  +MOVJ EC00435 VJ=100.00
SMOVL C00436 BC00436 V=100.0  +MOVJ EC00436
SMOVL C00437 BC00437 V=100.0 PL=0  +MOVJ EC00437
SREFP 1 C00438 BC00438  +REFP EC00438
SREFP 2 C00439 BC00439  +REFP EC00439
MACRO1 MJ#(0) ARGF0
ARCON
SMOVL C00440 BC00440 V=10.0  +MOVJ EC00440
ARCOF
SMOVL C00441 BC00441 V=400.0  +MOVJ EC00441
SMOVL C00442 BC00442 V=1000.0  +MOVJ EC00442
SSFTOF
MOVJ C00443 BC00443 VJ=100.00  +MOVJ EC00443 VJ=100.00
MOVJ C00444 BC00444 VJ=100.00  +MOVJ EC00444 VJ=100.00
MOVJ C00445 BC00445 VJ=100.00  +MOVJ EC00445 VJ=100.00
'
'Path W1682
SSFTOF
SSFTON P023
SMOVL C00446 BC00446 V=100.0  +MOVJ EC00446
SMOVL C00447 BC00447 V=100.0 PL=0  +MOVJ EC00447
SREFP 1 C00448 BC00448  +REFP EC00448
SREFP 2 C00449 BC00449  +REFP EC00449
MACRO1 MJ#(0) ARGF0
ARCON
SMOVL C00450 BC00450 V=10.0  +MOVJ EC00450
SMOVL C00451 BC00451 V=10.0  +MOVJ EC00451
SMOVL C00452 BC00452 V=10.0  +MOVJ EC00452
ARCOF
SMOVL C00453 BC00453 V=400.0  +MOVJ EC00453
SSFTOF
MOVJ C00454 BC00454 VJ=100.00  +MOVJ EC00454 VJ=100.00
'Path W1683
SSFTOF
SSFTON P023
MOVJ C00455 BC00455 VJ=100.00  +MOVJ EC00455 VJ=100.00
SMOVL C00456 BC00456 V=100.0  +MOVJ EC00456
SMOVL C00457 BC00457 V=100.0 PL=0  +MOVJ EC00457
SREFP 1 C00458 BC00458  +REFP EC00458
SREFP 2 C00459 BC00459  +REFP EC00459
MACRO1 MJ#(0) ARGF0
ARCON
SMOVL C00460 BC00460 V=10.0  +MOVJ EC00460
SMOVL C00461 BC00461 V=10.0  +MOVJ EC00461
SMOVL C00462 BC00462 V=10.0  +MOVJ EC00462
ARCOF
SMOVL C00463 BC00463 V=400.0  +MOVJ EC00463
SMOVL C00464 BC00464 V=1000.0  +MOVJ EC00464
SSFTOF
MOVJ C00465 BC00465 VJ=100.00  +MOVJ EC00465 VJ=100.00
'
'Path W1684
SSFTOF
SSFTON P024
MOVJ C00466 BC00466 VJ=100.00  +MOVJ EC00466 VJ=100.00
SMOVL C00467 BC00467 V=100.0  +MOVJ EC00467
SMOVL C00468 BC00468 V=100.0 PL=0  +MOVJ EC00468
SREFP 1 C00469 BC00469  +REFP EC00469
SREFP 2 C00470 BC00470  +REFP EC00470
MACRO1 MJ#(0) ARGF0
ARCON
SMOVL C00471 BC00471 V=10.0  +MOVJ EC00471
SMOVL C00472 BC00472 V=10.0  +MOVJ EC00472
SMOVL C00473 BC00473 V=10.0  +MOVJ EC00473
ARCOF
SMOVL C00474 BC00474 V=400.0  +MOVJ EC00474
SMOVL C00475 BC00475 V=1000.0  +MOVJ EC00475
SSFTOF
'Path W1685
SSFTOF
SSFTON P025
MOVJ C00476 BC00476 VJ=100.00  +MOVJ EC00476 VJ=100.00
SMOVL C00477 BC00477 V=100.0  +MOVJ EC00477
SMOVL C00478 BC00478 V=100.0 PL=0  +MOVJ EC00478
SREFP 1 C00479 BC00479  +REFP EC00479
SREFP 2 C00480 BC00480  +REFP EC00480
MACRO1 MJ#(0) ARGF0
ARCON
SMOVL C00481 BC00481 V=10.0  +MOVJ EC00481
SMOVL C00482 BC00482 V=10.0  +MOVJ EC00482
SMOVL C00483 BC00483 V=10.0  +MOVJ EC00483
ARCOF
SMOVL C00484 BC00484 V=400.0  +MOVJ EC00484
SMOVL C00485 BC00485 V=1000.0  +MOVJ EC00485
SSFTOF
'
MOVJ C00486 BC00486 VJ=100.00  +MOVJ EC00486 VJ=100.00
MOVJ C00487 BC00487 VJ=100.00  +MOVJ EC00487 VJ=100.00
MOVJ C00488 BC00488 VJ=100.00  +MOVJ EC00488 VJ=100.00
MOVJ C00489 BC00489 VJ=100.00  +MOVJ EC00489 VJ=100.00
'Path W1686
SSFTOF
SSFTON P024
MOVJ C00490 BC00490 VJ=100.00  +MOVJ EC00490 VJ=100.00
SMOVL C00491 BC00491 V=100.0 PL=0  +MOVJ EC00491
SREFP 1 C00492 BC00492  +REFP EC00492
SREFP 2 C00493 BC00493  +REFP EC00493
MACRO1 MJ#(0) ARGF0
ARCON
SMOVL C00494 BC00494 V=10.0  +MOVJ EC00494
SMOVL C00495 BC00495 V=10.0  +MOVJ EC00495
SMOVL C00496 BC00496 V=10.0  +MOVJ EC00496
ARCOF
SMOVL C00497 BC00497 V=400.0  +MOVJ EC00497
SSFTOF
MOVJ C00498 BC00498 VJ=100.00  +MOVJ EC00498 VJ=100.00
'Path W1687
SSFTOF
SSFTON P025
MOVJ C00499 BC00499 VJ=100.00  +MOVJ EC00499 VJ=100.00
SMOVL C00500 BC00500 V=100.0  +MOVJ EC00500
SMOVL C00501 BC00501 V=100.0 PL=0  +MOVJ EC00501
SREFP 1 C00502 BC00502  +REFP EC00502
SREFP 2 C00503 BC00503  +REFP EC00503
MACRO1 MJ#(0) ARGF0
ARCON
SMOVL C00504 BC00504 V=10.0  +MOVJ EC00504
SMOVL C00505 BC00505 V=10.0  +MOVJ EC00505
SMOVL C00506 BC00506 V=10.0  +MOVJ EC00506
ARCOF
SMOVL C00507 BC00507 V=400.0  +MOVJ EC00507
SMOVL C00508 BC00508 V=1000.0  +MOVJ EC00508
SSFTOF
MOVJ C00509 BC00509 VJ=100.00  +MOVJ EC00509 VJ=100.00
MOVJ C00510 BC00510 VJ=100.00  +MOVJ EC00510 VJ=100.00
'
MOVJ C00511 BC00511 VJ=100.00  +MOVJ EC00511 VJ=100.00
MOVJ C00512 BC00512 VJ=100.00  +MOVJ EC00512 VJ=100.00
MOVJ C00513 BC00513 VJ=100.00  +MOVJ EC00513 VJ=100.00
'Path W1688
SSFTOF
SSFTON P026
MOVJ C00514 BC00514 VJ=100.00  +MOVJ EC00514 VJ=100.00
SMOVL C00515 BC00515 V=100.0  +MOVJ EC00515
SMOVL C00516 BC00516 V=100.0 PL=0  +MOVJ EC00516
SREFP 1 C00517 BC00517  +REFP EC00517
SREFP 2 C00518 BC00518  +REFP EC00518
MACRO1 MJ#(0) ARGF0
ARCON
SMOVL C00519 BC00519 V=10.0  +MOVJ EC00519
SMOVL C00520 BC00520 V=10.0  +MOVJ EC00520
SMOVL C00521 BC00521 V=10.0  +MOVJ EC00521
ARCOF
SMOVL C00522 BC00522 V=400.0  +MOVJ EC00522
SMOVL C00523 BC00523 V=1000.0  +MOVJ EC00523
SSFTOF
'Path W1689
SSFTOF
SSFTON P027
MOVJ C00524 BC00524 VJ=100.00  +MOVJ EC00524 VJ=100.00
SMOVL C00525 BC00525 V=100.0  +MOVJ EC00525
SMOVL C00526 BC00526 V=100.0 PL=0  +MOVJ EC00526
SREFP 1 C00527 BC00527  +REFP EC00527
SREFP 2 C00528 BC00528  +REFP EC00528
MACRO1 MJ#(0) ARGF0
ARCON
SMOVL C00529 BC00529 V=10.0  +MOVJ EC00529
SMOVL C00530 BC00530 V=10.0  +MOVJ EC00530
SMOVL C00531 BC00531 V=10.0  +MOVJ EC00531
ARCOF
SMOVL C00532 BC00532 V=400.0  +MOVJ EC00532
SMOVL C00533 BC00533 V=1000.0  +MOVJ EC00533
SSFTOF
MOVJ C00534 BC00534 VJ=100.00  +MOVJ EC00534 VJ=100.00
MOVJ C00535 BC00535 VJ=100.00  +MOVJ EC00535 VJ=100.00
MOVJ C00536 BC00536 VJ=100.00  +MOVJ EC00536 VJ=100.00
MOVJ C00537 BC00537 VJ=100.00  +MOVJ EC00537 VJ=100.00
MOVJ C00538 BC00538 VJ=100.00  +MOVJ EC00538 VJ=100.00
'66
'jakie searche do takicj spoin?
'Path W1973
SSFTOF
MOVJ C00539 BC00539 VJ=100.00  +MOVJ EC00539 VJ=100.00
MOVL C00540 BC00540 V=100.0  +MOVJ EC00540 VJ=100.00
SMOVL C00541 BC00541 V=100.0 PL=0  +MOVJ EC00541
SREFP 1 C00542 BC00542  +REFP EC00542
SREFP 2 C00543 BC00543  +REFP EC00543
MACRO1 MJ#(0) ARGF0
ARCON
SMOVL C00544 BC00544 V=10.0  +MOVJ EC00544
ARCOF
MOVL C00545 BC00545 V=400.0  +MOVJ EC00545 VJ=100.00
MOVL C00546 BC00546 V=1000.0  +MOVJ EC00546 VJ=100.00
'brak dostÄpu do jednej spoiny
MOVJ C00547 BC00547 VJ=100.00  +MOVJ EC00547 VJ=100.00
'Path W1691
SSFTOF
MOVJ C00548 BC00548 VJ=100.00  +MOVJ EC00548 VJ=100.00
MOVL C00549 BC00549 V=100.0  +MOVJ EC00549 VJ=100.00
SMOVL C00550 BC00550 V=100.0 PL=0  +MOVJ EC00550
SREFP 1 C00551 BC00551  +REFP EC00551
SREFP 2 C00552 BC00552  +REFP EC00552
MACRO1 MJ#(0) ARGF0
ARCON
SMOVL C00553 BC00553 V=10.0  +MOVJ EC00553
ARCOF
MOVL C00554 BC00554 V=400.0  +MOVJ EC00554 VJ=100.00
MOVL C00555 BC00555 V=1000.0  +MOVJ EC00555 VJ=100.00
'Path W1692
SSFTOF
MOVJ C00556 BC00556 VJ=100.00  +MOVJ EC00556 VJ=100.00
MOVL C00557 BC00557 V=100.0  +MOVJ EC00557 VJ=100.00
SMOVL C00558 BC00558 V=100.0 PL=0  +MOVJ EC00558
SREFP 1 C00559 BC00559  +REFP EC00559
SREFP 2 C00560 BC00560  +REFP EC00560
MACRO1 MJ#(0) ARGF0
ARCON
SMOVL C00561 BC00561 V=10.0  +MOVJ EC00561
ARCOF
MOVL C00562 BC00562 V=400.0  +MOVJ EC00562 VJ=100.00
MOVL C00563 BC00563 V=1000.0  +MOVJ EC00563 VJ=100.00
MOVJ C00564 BC00564 VJ=100.00  +MOVJ EC00564 VJ=100.00
'Path W1693
SSFTOF
MOVJ C00565 BC00565 VJ=100.00  +MOVJ EC00565 VJ=100.00
MOVL C00566 BC00566 V=100.0  +MOVJ EC00566 VJ=100.00
SMOVL C00567 BC00567 V=100.0 PL=0  +MOVJ EC00567
SREFP 1 C00568 BC00568  +REFP EC00568
SREFP 2 C00569 BC00569  +REFP EC00569
MACRO1 MJ#(0) ARGF0
ARCON
SMOVL C00570 BC00570 V=10.0  +MOVJ EC00570
ARCOF
MOVL C00571 BC00571 V=400.0  +MOVJ EC00571 VJ=100.00
MOVL C00572 BC00572 V=1000.0  +MOVJ EC00572 VJ=100.00
'Path W1694
SSFTOF
MOVJ C00573 BC00573 VJ=100.00  +MOVJ EC00573 VJ=100.00
MOVL C00574 BC00574 V=100.0  +MOVJ EC00574 VJ=100.00
SMOVL C00575 BC00575 V=100.0 PL=0  +MOVJ EC00575
SREFP 1 C00576 BC00576  +REFP EC00576
SREFP 2 C00577 BC00577  +REFP EC00577
MACRO1 MJ#(0) ARGF0
ARCON
SMOVL C00578 BC00578 V=10.0  +MOVJ EC00578
ARCOF
MOVL C00579 BC00579 V=400.0  +MOVJ EC00579 VJ=100.00
MOVL C00580 BC00580 V=1000.0  +MOVJ EC00580 VJ=100.00
'Path W1695
SSFTOF
MOVJ C00581 BC00581 VJ=100.00  +MOVJ EC00581 VJ=100.00
MOVL C00582 BC00582 V=100.0  +MOVJ EC00582 VJ=100.00
SMOVL C00583 BC00583 V=100.0 PL=0  +MOVJ EC00583
SREFP 1 C00584 BC00584  +REFP EC00584
SREFP 2 C00585 BC00585  +REFP EC00585
MACRO1 MJ#(0) ARGF0
ARCON
SMOVL C00586 BC00586 V=10.0  +MOVJ EC00586
ARCOF
MOVL C00587 BC00587 V=400.0  +MOVJ EC00587 VJ=100.00
MOVL C00588 BC00588 V=1000.0  +MOVJ EC00588 VJ=100.00
'Path W1696
SSFTOF
MOVJ C00589 BC00589 VJ=100.00  +MOVJ EC00589 VJ=100.00
MOVL C00590 BC00590 V=100.0  +MOVJ EC00590 VJ=100.00
SMOVL C00591 BC00591 V=100.0 PL=0  +MOVJ EC00591
SREFP 1 C00592 BC00592  +REFP EC00592
SREFP 2 C00593 BC00593  +REFP EC00593
MACRO1 MJ#(0) ARGF0
ARCON
SMOVL C00594 BC00594 V=10.0  +MOVJ EC00594
ARCOF
MOVL C00595 BC00595 V=400.0  +MOVJ EC00595 VJ=100.00
MOVL C00596 BC00596 V=1000.0  +MOVJ EC00596 VJ=100.00
'67
'jakie searche do takicj spoin?
'Path W1697
SSFTOF
MOVJ C00597 BC00597 VJ=100.00  +MOVJ EC00597 VJ=100.00
MOVL C00598 BC00598 V=100.0  +MOVJ EC00598 VJ=100.00
SMOVL C00599 BC00599 V=100.0 PL=0  +MOVJ EC00599
SREFP 1 C00600 BC00600  +REFP EC00600
SREFP 2 C00601 BC00601  +REFP EC00601
MACRO1 MJ#(0) ARGF0
ARCON
SMOVL C00602 BC00602 V=10.0  +MOVJ EC00602
SMOVL C00603 BC00603 V=10.0  +MOVJ EC00603
SMOVL C00604 BC00604 V=10.0  +MOVJ EC00604
ARCOF
MOVL C00605 BC00605 V=400.0  +MOVJ EC00605 VJ=100.00
MOVL C00606 BC00606 V=1000.0  +MOVJ EC00606 VJ=100.00
'Path W1698
SSFTOF
MOVJ C00607 BC00607 VJ=100.00  +MOVJ EC00607 VJ=100.00
MOVL C00608 BC00608 V=100.0  +MOVJ EC00608 VJ=100.00
SMOVL C00609 BC00609 V=100.0 PL=0  +MOVJ EC00609
SREFP 1 C00610 BC00610  +REFP EC00610
SREFP 2 C00611 BC00611  +REFP EC00611
MACRO1 MJ#(0) ARGF0
ARCON
SMOVL C00612 BC00612 V=10.0  +MOVJ EC00612
SMOVL C00613 BC00613 V=10.0  +MOVJ EC00613
SMOVL C00614 BC00614 V=10.0  +MOVJ EC00614
ARCOF
MOVL C00615 BC00615 V=400.0  +MOVJ EC00615 VJ=100.00
MOVL C00616 BC00616 V=1000.0  +MOVJ EC00616 VJ=100.00
'68,69
MOVJ C00617 BC00617 VJ=100.00  +MOVJ EC00617 VJ=100.00
'Path W1699
SSFTOF
SSFTON P030
MOVJ C00618 BC00618 VJ=100.00  +MOVJ EC00618 VJ=100.00
SMOVL C00619 BC00619 V=100.0  +MOVJ EC00619
SMOVL C00620 BC00620 V=100.0 PL=0  +MOVJ EC00620
SREFP 1 C00621 BC00621  +REFP EC00621
SREFP 2 C00622 BC00622  +REFP EC00622
MACRO1 MJ#(0) ARGF0
ARCON
SSFTON P029
SMOVL C00623 BC00623 V=10.0  +MOVJ EC00623
SMOVL C00624 BC00624 V=10.0  +MOVJ EC00624
SSFTON P028
SMOVL C00625 BC00625 V=10.0  +MOVJ EC00625
ARCOF
SMOVL C00626 BC00626 V=400.0  +MOVJ EC00626
SMOVL C00627 BC00627 V=1000.0  +MOVJ EC00627
SSFTOF
MOVJ C00628 BC00628 VJ=100.00  +MOVJ EC00628 VJ=100.00
MOVJ C00629 BC00629 VJ=100.00  +MOVJ EC00629 VJ=100.00
MOVJ C00630 BC00630 VJ=100.00  +MOVJ EC00630 VJ=100.00
MOVJ C00631 BC00631 VJ=100.00  +MOVJ EC00631 VJ=100.00
'Path W1700
SSFTOF
SSFTON P031
MOVJ C00632 BC00632 VJ=100.00  +MOVJ EC00632 VJ=100.00
SMOVL C00633 BC00633 V=100.0  +MOVJ EC00633
SMOVL C00634 BC00634 V=100.0 PL=0  +MOVJ EC00634
SREFP 1 C00635 BC00635  +REFP EC00635
SREFP 2 C00636 BC00636  +REFP EC00636
MACRO1 MJ#(0) ARGF0
ARCON
SMOVL C00637 BC00637 V=10.0  +MOVJ EC00637
SMOVL C00638 BC00638 V=10.0  +MOVJ EC00638
SMOVL C00639 BC00639 V=10.0  +MOVJ EC00639
ARCOF
SMOVL C00640 BC00640 V=400.0  +MOVJ EC00640
SMOVL C00641 BC00641 V=1000.0  +MOVJ EC00641
SSFTOF
END
